C05458=1037.244,431.562,355.242,175.283,46.593,159.539
C05459=1037.232,431.317,355.292,175.268,46.586,159.535
C05460=1037.220,431.072,355.342,175.254,46.579,159.532
C05461=1037.208,430.829,355.393,175.240,46.572,159.528
C05462=1037.196,430.584,355.443,175.226,46.565,159.524
C05463=1037.184,430.339,355.494,175.213,46.558,159.521
C05464=1037.173,430.095,355.544,175.199,46.551,159.517
C05465=1037.161,429.850,355.594,175.184,46.544,159.513
C05466=1037.149,429.606,355.644,175.171,46.537,159.510
C05467=1037.138,429.360,355.694,175.157,46.530,159.506
C05468=1037.125,429.116,355.744,175.144,46.523,159.502
C05469=1037.114,428.871,355.793,175.130,46.516,159.499
C05470=1037.103,428.626,355.844,175.117,46.509,159.495
C05471=1037.091,428.382,355.894,175.103,46.503,159.492
C05472=1037.080,428.137,355.944,175.090,46.495,159.488
C05473=1037.068,427.892,355.994,175.076,46.489,159.485
C05474=1037.056,427.648,356.043,175.063,46.482,159.481
C05475=1037.044,427.402,356.093,175.049,46.475,159.478
C05476=1037.033,427.157,356.142,175.036,46.468,159.474
C05477=1037.022,426.913,356.192,175.023,46.462,159.471
C05478=1037.010,426.668,356.241,175.010,46.455,159.467
C05479=1036.998,426.423,356.290,174.997,46.448,159.464
C05480=1036.987,426.178,356.339,174.984,46.442,159.460
C05481=1036.975,425.933,356.389,174.970,46.435,159.457
C05482=1036.963,425.689,356.439,174.957,46.428,159.453
C05483=1036.952,425.444,356.488,174.944,46.422,159.450
C05484=1036.941,425.199,356.537,174.932,46.415,159.447
C05485=1036.930,424.953,356.585,174.919,46.409,159.443
C05486=1036.918,424.709,356.634,174.905,46.402,159.440
C05487=1036.907,424.464,356.684,174.892,46.395,159.436
C05488=1036.896,424.219,356.733,174.880,46.389,159.433
C05489=1036.884,423.974,356.782,174.867,46.383,159.430
C05490=1036.873,423.730,356.831,174.855,46.376,159.427
C05491=1036.861,423.484,356.879,174.842,46.370,159.423
C05492=1036.850,423.239,356.928,174.830,46.364,159.420
C05493=1036.839,423.000,356.976,174.817,46.357,159.417
C05494=1036.828,422.760,357.023,174.805,46.351,159.414
C05495=1036.817,422.521,357.070,174.793,46.345,159.411
C05496=1036.806,422.281,357.118,174.781,46.339,159.408
C05497=1036.795,422.041,357.165,174.769,46.333,159.404
C05498=1036.784,421.802,357.212,174.756,46.326,159.401
C05499=1036.774,421.562,357.259,174.745,46.320,159.398
C05500=1036.763,421.322,357.307,174.732,46.314,159.395
C05501=1036.752,421.077,357.355,174.720,46.308,159.392
C05502=1036.740,420.833,357.402,174.708,46.302,159.389
C05503=1036.729,420.588,357.451,174.696,46.296,159.386
C05504=1036.718,420.343,357.500,174.684,46.290,159.382
C05505=1036.708,420.097,357.547,174.672,46.283,159.379
C05506=1036.697,419.852,357.595,174.659,46.278,159.376
C05507=1036.685,419.607,357.644,174.648,46.271,159.373
C05508=1036.675,419.362,357.691,174.636,46.265,159.370
C05509=1036.664,419.117,357.740,174.623,46.259,159.367
C05510=1036.653,418.871,357.788,174.612,46.253,159.364
C05511=1036.642,418.626,357.835,174.600,46.247,159.361
C05512=1036.631,418.381,357.883,174.589,46.241,159.358
C05513=1036.620,418.136,357.931,174.576,46.235,159.355
C05514=1036.610,417.891,357.978,174.565,46.229,159.352
C05515=1036.599,417.646,358.026,174.553,46.223,159.349
C05516=1036.589,417.400,358.074,174.541,46.217,159.346
C05517=1036.577,417.155,358.121,174.530,46.211,159.343
C05518=1036.567,416.910,358.169,174.518,46.205,159.340
C05519=1036.556,416.664,358.216,174.507,46.200,159.337
C05520=1036.545,416.419,358.263,174.496,46.194,159.334
C05521=1036.535,416.174,358.311,174.484,46.188,159.331
C05522=1036.523,415.929,358.358,174.473,46.182,159.328
C05523=1036.513,415.683,358.405,174.461,46.177,159.325
C05524=1036.503,415.438,358.452,174.450,46.171,159.322
C05525=1036.491,415.192,358.499,174.439,46.165,159.320
C05526=1036.481,414.947,358.546,174.427,46.160,159.317
C05527=1036.470,414.702,358.593,174.416,46.154,159.314
C05528=1036.460,414.457,358.640,174.405,46.148,159.311
C05529=1036.450,414.212,358.687,174.393,46.142,159.308
C05530=1036.438,413.965,358.734,174.382,46.137,159.305
C05531=1036.428,413.720,358.781,174.371,46.131,159.303
C05532=1036.417,413.475,358.827,174.360,46.126,159.300
C05533=1036.407,413.230,358.875,174.349,46.120,159.297
C05534=1036.397,412.984,358.921,174.337,46.114,159.294
C05535=1036.386,412.739,358.968,174.327,46.109,159.291
C05536=1036.376,412.494,359.015,174.316,46.103,159.289
C05537=1036.365,412.248,359.061,174.305,46.098,159.286
C05538=1036.355,412.003,359.108,174.294,46.093,159.283
C05539=1036.345,411.757,359.155,174.284,46.087,159.281
C05540=1036.334,411.512,359.201,174.272,46.082,159.278
C05541=1036.325,411.266,359.248,174.261,46.076,159.275
C05542=1036.314,411.020,359.294,174.250,46.070,159.272
C05543=1036.303,410.775,359.340,174.240,46.065,159.270
C05544=1036.293,410.529,359.386,174.229,46.060,159.267
C05545=1036.283,410.285,359.432,174.218,46.055,159.264
C05546=1036.272,410.039,359.478,174.208,46.049,159.262
C05547=1036.262,409.793,359.524,174.197,46.044,159.259
C05548=1036.252,409.547,359.571,174.186,46.039,159.256
C05549=1036.241,409.302,359.617,174.176,46.034,159.254
C05550=1036.231,409.057,359.662,174.165,46.028,159.251
C05551=1036.221,408.811,359.707,174.155,46.023,159.249
C05552=1036.211,408.565,359.754,174.145,46.018,159.246
C05553=1036.201,408.330,359.798,174.135,46.013,159.244
C05554=1036.192,408.095,359.841,174.124,46.008,159.241
C05555=1036.181,407.860,359.886,174.115,46.003,159.239
C05556=1036.172,407.624,359.929,174.105,45.998,159.236
C05557=1036.162,407.390,359.972,174.095,45.993,159.234
C05558=1036.152,407.155,360.016,174.085,45.988,159.231
C05559=1036.144,406.919,360.060,174.076,45.983,159.229
C05560=1036.133,406.683,360.104,174.065,45.979,159.227
C05561=1036.123,406.439,360.150,174.056,45.973,159.224
C05562=1036.113,406.192,360.195,174.045,45.968,159.222
C05563=1036.103,405.947,360.240,174.035,45.963,159.219
C05564=1036.093,405.701,360.286,174.025,45.959,159.217
C05565=1036.084,405.455,360.331,174.015,45.953,159.214
C05566=1036.074,405.211,360.377,174.005,45.948,159.212
C05567=1036.063,404.964,360.422,173.995,45.944,159.209
C05568=1036.054,404.719,360.467,173.985,45.938,159.207
C05569=1036.044,404.474,360.513,173.975,45.933,159.204
C05570=1036.034,404.227,360.558,173.964,45.929,159.202
C05571=1036.024,403.982,360.603,173.955,45.923,159.199
C05572=1036.015,403.736,360.648,173.945,45.919,159.197
C05573=1036.005,403.490,360.693,173.936,45.914,159.195
C05574=1035.995,403.244,360.738,173.925,45.909,159.192
C05575=1035.986,402.999,360.783,173.916,45.904,159.190
C05576=1035.976,402.753,360.828,173.906,45.899,159.188
C05577=1035.966,402.508,360.873,173.896,45.894,159.185
C05578=1035.956,402.262,360.918,173.886,45.889,159.183
C05579=1035.946,402.016,360.963,173.877,45.885,159.181
C05580=1035.936,401.771,361.007,173.867,45.880,159.178
C05581=1035.927,401.525,361.052,173.858,45.875,159.176
C05582=1035.917,401.279,361.096,173.848,45.871,159.174
C05583=1035.908,401.033,361.141,173.838,45.866,159.171
C05584=1035.898,400.788,361.186,173.828,45.861,159.169
C05585=1035.889,400.542,361.230,173.819,45.856,159.167
C05586=1035.879,400.296,361.275,173.809,45.852,159.164
C05587=1035.869,400.050,361.319,173.800,45.848,159.162
C05588=1035.860,399.805,361.364,173.791,45.843,159.160
C05589=1035.850,399.558,361.408,173.781,45.838,159.158
C05590=1035.841,399.313,361.453,173.772,45.833,159.155
C05591=1035.830,399.067,361.496,173.763,45.829,159.153
C05592=1035.821,398.822,361.541,173.753,45.825,159.151
C05593=1035.811,398.575,361.585,173.743,45.820,159.149
C05594=1035.802,398.329,361.629,173.735,45.815,159.146
C05595=1035.792,398.083,361.673,173.724,45.811,159.144
C05596=1035.783,397.838,361.717,173.716,45.807,159.142
C05597=1035.773,397.593,361.761,173.707,45.802,159.140
C05598=1035.764,397.346,361.806,173.697,45.798,159.138
C05599=1035.754,397.100,361.850,173.688,45.793,159.135
C05600=1035.744,396.854,361.893,173.679,45.789,159.133
C05601=1035.735,396.609,361.937,173.670,45.784,159.131
C05602=1035.726,396.363,361.981,173.661,45.780,159.129
C05603=1035.717,396.117,362.025,173.651,45.776,159.127
C05604=1035.706,395.871,362.069,173.642,45.772,159.125
C05605=1035.698,395.626,362.112,173.633,45.767,159.122
C05606=1035.688,395.379,362.157,173.624,45.762,159.120
C05607=1035.679,395.133,362.200,173.615,45.758,159.118
C05608=1035.670,394.888,362.243,173.606,45.754,159.116
C05609=1035.660,394.641,362.287,173.597,45.750,159.114
C05610=1035.651,394.396,362.331,173.588,45.745,159.112
C05611=1035.642,394.150,362.374,173.579,45.741,159.110
C05612=1035.632,393.903,362.418,173.570,45.737,159.108
C05613=1035.623,393.678,362.457,173.563,45.733,159.106
C05614=1035.616,393.453,362.497,173.554,45.729,159.104
C05615=1035.607,393.228,362.536,173.545,45.725,159.102
C05616=1035.598,393.003,362.576,173.538,45.722,159.100
C05617=1035.590,392.778,362.616,173.530,45.718,159.098
C05618=1035.581,392.553,362.655,173.522,45.714,159.097
C05619=1035.573,392.328,362.695,173.514,45.710,159.095
C05620=1035.565,392.103,362.735,173.506,45.706,159.093
C05621=1035.555,391.857,362.777,173.497,45.702,159.091
C05622=1035.546,391.611,362.821,173.489,45.698,159.089
C05623=1035.537,391.366,362.864,173.480,45.694,159.087
C05624=1035.528,391.120,362.907,173.471,45.690,159.085
C05625=1035.519,390.873,362.950,173.462,45.686,159.083
C05626=1035.510,390.627,362.993,173.454,45.682,159.081
C05627=1035.501,390.380,363.036,173.445,45.678,159.079
C05628=1035.491,390.135,363.078,173.436,45.674,159.077
C05629=1035.482,389.889,363.121,173.428,45.670,159.075
C05630=1035.473,389.642,363.164,173.419,45.667,159.073
C05631=1035.464,389.396,363.207,173.412,45.662,159.071
C05632=1035.455,389.150,363.250,173.403,45.658,159.069
C05633=1035.446,388.905,363.292,173.394,45.654,159.067
C05634=1035.436,388.658,363.335,173.386,45.651,159.065
C05635=1035.428,388.412,363.378,173.377,45.647,159.063
C05636=1035.419,388.166,363.420,173.369,45.642,159.061
C05637=1035.410,387.920,363.463,173.361,45.638,159.060
C05638=1035.401,387.674,363.505,173.353,45.635,159.058
C05639=1035.391,387.427,363.548,173.344,45.631,159.056
C05640=1035.383,387.181,363.591,173.335,45.627,159.054
C05641=1035.374,386.935,363.633,173.327,45.623,159.052
C05642=1035.365,386.689,363.675,173.320,45.620,159.050
C05643=1035.356,386.443,363.717,173.311,45.616,159.048
C05644=1035.346,386.197,363.759,173.303,45.612,159.046
C05645=1035.337,385.950,363.801,173.294,45.608,159.045
C05646=1035.328,385.704,363.844,173.287,45.605,159.043
C05647=1035.319,385.458,363.886,173.278,45.601,159.041
C05648=1035.311,385.211,363.928,173.270,45.597,159.039
C05649=1035.301,384.966,363.970,173.261,45.594,159.037
C05650=1035.292,384.719,364.012,173.254,45.590,159.036
C05651=1035.283,384.473,364.054,173.245,45.586,159.034
C05652=1035.274,384.226,364.095,173.237,45.583,159.032
C05653=1035.265,383.981,364.138,173.230,45.579,159.030
C05654=1035.256,383.734,364.180,173.221,45.576,159.028
C05655=1035.248,383.488,364.222,173.213,45.572,159.027
C05656=1035.239,383.241,364.264,173.206,45.568,159.025
C05657=1035.230,382.995,364.305,173.197,45.565,159.023
C05658=1035.222,382.749,364.347,173.190,45.561,159.021
C05659=1035.213,382.503,364.388,173.181,45.557,159.019
C05660=1035.204,382.257,364.430,173.173,45.554,159.018
C05661=1035.195,382.010,364.472,173.166,45.551,159.016
C05662=1035.186,381.764,364.514,173.157,45.547,159.014
C05663=1035.177,381.517,364.555,173.150,45.543,159.012
C05664=1035.170,381.271,364.597,173.142,45.540,159.011
C05665=1035.161,381.025,364.639,173.135,45.537,159.009
C05666=1035.152,380.779,364.681,173.126,45.533,159.007
C05667=1035.143,380.532,364.722,173.119,45.529,159.006
C05668=1035.135,380.286,364.763,173.111,45.526,159.004
C05669=1035.126,380.040,364.805,173.104,45.523,159.002
C05670=1035.117,379.793,364.846,173.095,45.519,159.001
C05671=1035.108,379.547,364.888,173.088,45.516,158.999
C05672=1035.100,379.301,364.929,173.080,45.512,158.997
C05673=1035.085,378.885,364.999,173.067,45.506,158.994
C05674=1035.071,378.470,365.069,173.054,45.501,158.992
C05675=1035.057,378.055,365.138,173.042,45.495,158.989
C05676=1035.043,377.640,365.208,173.029,45.490,158.986
C05677=1035.033,377.393,365.248,173.021,45.487,158.984
C05678=1035.025,377.147,365.289,173.014,45.483,158.983
C05679=1035.017,376.900,365.330,173.005,45.480,158.981
C05680=1035.008,376.653,365.372,172.998,45.477,158.980
C05681=1035.000,376.407,365.412,172.991,45.473,158.978
C05682=1034.990,376.160,365.453,172.983,45.470,158.976
C05683=1034.982,375.914,365.493,172.976,45.467,158.975
C05684=1034.974,375.667,365.534,172.968,45.464,158.973
C05685=1034.965,375.421,365.576,172.961,45.461,158.972
C05686=1034.956,375.175,365.616,172.954,45.457,158.970
C05687=1034.948,374.929,365.657,172.946,45.455,158.968
C05688=1034.939,374.682,365.698,172.939,45.451,158.967
C05689=1034.931,374.435,365.738,172.932,45.448,158.965
C05690=1034.922,374.189,365.778,172.924,45.445,158.964
C05691=1034.914,373.942,365.819,172.916,45.442,158.962
C05692=1034.906,373.696,365.860,172.909,45.439,158.961
C05693=1034.897,373.449,365.901,172.902,45.436,158.959
C05694=1034.889,373.202,365.940,172.895,45.433,158.957
C05695=1034.881,372.956,365.981,172.887,45.430,158.956
C05696=1034.872,372.709,366.022,172.880,45.426,158.954
C05697=1034.863,372.463,366.062,172.873,45.423,158.953
C05698=1034.855,372.217,366.103,172.866,45.421,158.951
C05699=1034.847,371.969,366.143,172.858,45.418,158.950
C05700=1034.839,371.723,366.184,172.851,45.414,158.948
C05701=1034.830,371.477,366.224,172.844,45.411,158.947
C05702=1034.822,371.231,366.264,172.837,45.408,158.945
C05703=1034.814,370.983,366.304,172.830,45.405,158.944
C05704=1034.806,370.737,366.345,172.823,45.402,158.942
C05705=1034.797,370.490,366.384,172.815,45.400,158.941
C05706=1034.789,370.244,366.425,172.809,45.397,158.939
C05707=1034.781,369.998,366.466,172.802,45.394,158.938
C05708=1034.773,369.751,366.505,172.795,45.391,158.936
C05709=1034.764,369.503,366.545,172.788,45.388,158.935
C05710=1034.756,369.257,366.585,172.781,45.385,158.933
C05711=1034.748,369.011,366.625,172.774,45.382,158.932
C05712=1034.740,368.764,366.665,172.766,45.379,158.930
C05713=1034.731,368.518,366.705,172.759,45.377,158.929
C05714=1034.723,368.271,366.745,172.752,45.374,158.928
C05715=1034.714,368.024,366.784,172.745,45.371,158.926
C05716=1034.706,367.777,366.824,172.739,45.368,158.925
C05717=1034.698,367.531,366.864,172.732,45.366,158.924
C05718=1034.689,367.284,366.904,172.725,45.363,158.922
C05719=1034.681,367.037,366.943,172.718,45.360,158.921
C05720=1034.673,366.791,366.983,172.711,45.357,158.919
C05721=1034.665,366.544,367.023,172.704,45.354,158.918
C05722=1034.657,366.297,367.062,172.698,45.351,158.916
C05723=1034.648,366.051,367.101,172.691,45.349,158.915
C05724=1034.641,365.804,367.141,172.684,45.346,158.914
C05725=1034.632,365.557,367.181,172.677,45.343,158.912
C05726=1034.624,365.310,367.220,172.670,45.340,158.911
C05727=1034.616,365.064,367.260,172.664,45.338,158.910
C05728=1034.607,364.817,367.299,172.657,45.335,158.908
C05729=1034.595,364.422,367.362,172.646,45.331,158.906
C05730=1034.582,364.028,367.425,172.635,45.327,158.904
C05731=1034.569,363.633,367.488,172.624,45.322,158.902
C05732=1034.557,363.238,367.551,172.614,45.318,158.899
C05733=1034.548,362.991,367.591,172.607,45.316,158.898
C05734=1034.540,362.745,367.630,172.600,45.313,158.897
C05735=1034.533,362.498,367.669,172.593,45.310,158.895
C05736=1034.524,362.251,367.708,172.587,45.308,158.894
C05737=1034.516,362.005,367.747,172.580,45.306,158.893
C05738=1034.509,361.757,367.787,172.573,45.303,158.892
C05739=1034.501,361.511,367.826,172.567,45.300,158.890
C05740=1034.492,361.264,367.864,172.561,45.297,158.889
C05741=1034.484,361.017,367.903,172.554,45.295,158.888
C05742=1034.477,360.770,367.943,172.548,45.293,158.886
C05743=1034.468,360.523,367.982,172.541,45.290,158.885
C05744=1034.461,360.277,368.020,172.534,45.288,158.884
C05745=1034.452,360.030,368.059,172.528,45.285,158.882
C05746=1034.444,359.783,368.098,172.521,45.283,158.881
C05747=1034.436,359.536,368.136,172.515,45.280,158.880
C05748=1034.428,359.289,368.175,172.509,45.278,158.879
C05749=1034.420,359.042,368.214,172.502,45.276,158.877
C05750=1034.412,358.795,368.253,172.495,45.273,158.876
C05751=1034.404,358.549,368.291,172.489,45.271,158.875
C05752=1034.396,358.302,368.330,172.482,45.269,158.874
C05753=1034.388,358.055,368.368,172.477,45.266,158.873
C05754=1034.380,357.808,368.407,172.470,45.264,158.871
C05755=1034.372,357.561,368.445,172.463,45.261,158.870
C05756=1034.365,357.314,368.484,172.457,45.259,158.869
C05757=1034.357,357.067,368.523,172.451,45.257,158.868
C05758=1034.349,356.821,368.562,172.445,45.254,158.866
C05759=1034.341,356.574,368.600,172.438,45.252,158.865
C05760=1034.333,356.326,368.639,172.432,45.250,158.864
C05761=1034.325,356.080,368.677,172.426,45.248,158.863
C05762=1034.318,355.832,368.715,172.420,45.245,158.861
C05763=1034.310,355.586,368.753,172.413,45.243,158.860
C05764=1034.301,355.339,368.791,172.407,45.241,158.859
C05765=1034.294,355.092,368.830,172.401,45.238,158.858
C05766=1034.285,354.845,368.868,172.395,45.236,158.857
C05767=1034.278,354.598,368.906,172.388,45.234,158.855
C05768=1034.270,354.351,368.944,172.382,45.232,158.854
C05769=1034.263,354.104,368.983,172.376,45.229,158.853
C05770=1034.254,353.857,369.021,172.370,45.228,158.852
C05771=1034.246,353.610,369.058,172.363,45.225,158.851
C05772=1034.239,353.363,369.096,172.358,45.223,158.850
C05773=1034.231,353.116,369.135,172.351,45.221,158.848
C05774=1034.223,352.869,369.172,172.345,45.219,158.847
C05775=1034.215,352.622,369.211,172.339,45.217,158.846
C05776=1034.207,352.375,369.248,172.333,45.214,158.845
C05777=1034.200,352.129,369.286,172.326,45.212,158.844
C05778=1034.192,351.881,369.324,172.321,45.210,158.843
C05779=1034.184,351.634,369.362,172.314,45.208,158.842
C05780=1034.177,351.387,369.400,172.308,45.206,158.840
C05781=1034.169,351.140,369.438,172.303,45.204,158.839
C05782=1034.161,350.893,369.475,172.296,45.202,158.838
C05783=1034.153,350.647,369.514,172.291,45.199,158.837
C05784=1034.146,350.399,369.552,172.284,45.198,158.836
C05785=1034.134,350.011,369.611,172.275,45.194,158.834
C05786=1034.121,349.622,369.670,172.266,45.191,158.833
C05787=1034.110,349.233,369.729,172.256,45.188,158.831
C05788=1034.097,348.844,369.788,172.246,45.185,158.829
C05789=1034.090,348.597,369.826,172.241,45.183,158.828
C05790=1034.082,348.351,369.864,172.235,45.181,158.827
C05791=1034.075,348.104,369.901,172.229,45.179,158.826
C05792=1034.067,347.857,369.938,172.223,45.177,158.825
C05793=1034.059,347.609,369.976,172.217,45.175,158.824
C05794=1034.051,347.362,370.013,172.211,45.173,158.823
C05795=1034.044,347.115,370.050,172.205,45.171,158.822
C05796=1034.036,346.868,370.087,172.200,45.169,158.820
C05797=1034.028,346.621,370.125,172.193,45.167,158.819
C05798=1034.021,346.374,370.162,172.188,45.165,158.818
C05799=1034.013,346.127,370.199,172.182,45.163,158.817
C05800=1034.005,345.880,370.237,172.176,45.161,158.816
C05801=1033.997,345.633,370.274,172.170,45.160,158.815
C05802=1033.990,345.386,370.312,172.165,45.158,158.814
C05803=1033.982,345.138,370.348,172.158,45.156,158.813
C05804=1033.975,344.891,370.385,172.153,45.154,158.812
C05805=1033.967,344.644,370.422,172.147,45.152,158.811
C05806=1033.960,344.397,370.460,172.142,45.151,158.810
C05807=1033.952,344.150,370.497,172.136,45.149,158.809
C05808=1033.945,343.902,370.534,172.130,45.147,158.808
C05809=1033.936,343.603,370.578,172.124,45.145,158.807
C05810=1033.926,343.303,370.624,172.116,45.143,158.806
C05811=1033.917,343.003,370.669,172.109,45.140,158.804
C05812=1033.908,342.703,370.713,172.103,45.138,158.803
C05813=1033.901,342.456,370.750,172.097,45.136,158.802
C05814=1033.893,342.209,370.786,172.091,45.134,158.801
C05815=1033.886,341.962,370.824,172.085,45.133,158.800
C05816=1033.878,341.715,370.861,172.080,45.131,158.799
C05817=1033.871,341.467,370.897,172.075,45.129,158.798
C05818=1033.863,341.220,370.935,172.068,45.127,158.797
C05819=1033.856,340.973,370.971,172.063,45.126,158.796
C05820=1033.849,340.725,371.008,172.057,45.124,158.795
C05821=1033.841,340.478,371.045,172.052,45.123,158.794
C05822=1033.833,340.231,371.081,172.046,45.120,158.793
C05823=1033.825,339.984,371.118,172.040,45.119,158.792
C05824=1033.818,339.737,371.154,172.035,45.118,158.791
C05825=1033.811,339.490,371.190,172.029,45.116,158.790
C05826=1033.803,339.242,371.227,172.024,45.114,158.789
C05827=1033.795,338.995,371.264,172.019,45.113,158.789
C05828=1033.788,338.748,371.300,172.012,45.111,158.787
C05829=1033.780,338.500,371.336,172.007,45.109,158.787
C05830=1033.774,338.253,371.372,172.002,45.108,158.786
C05831=1033.766,338.007,371.409,171.996,45.107,158.785
C05832=1033.758,337.759,371.446,171.991,45.104,158.784
C05833=1033.750,337.512,371.482,171.986,45.103,158.783
C05834=1033.743,337.265,371.518,171.980,45.102,158.782
C05835=1033.736,337.017,371.554,171.975,45.100,158.781
C05836=1033.729,336.770,371.591,171.969,45.098,158.780
C05837=1033.721,336.522,371.627,171.964,45.096,158.779
C05838=1033.714,336.275,371.663,171.958,45.095,158.778
C05839=1033.706,336.028,371.699,171.953,45.094,158.777
C05840=1033.699,335.781,371.735,171.948,45.092,158.776
C05841=1033.689,335.442,371.785,171.940,45.090,158.775
C05842=1033.679,335.103,371.835,171.933,45.088,158.774
C05843=1033.669,334.764,371.884,171.925,45.086,158.773
C05844=1033.659,334.424,371.934,171.918,45.084,158.771
C05845=1033.651,334.177,371.970,171.913,45.082,158.770
C05846=1033.644,333.930,372.006,171.907,45.081,158.770
C05847=1033.636,333.682,372.042,171.902,45.079,158.769
C05848=1033.629,333.434,372.077,171.896,45.078,158.768
C05849=1033.622,333.188,372.113,171.892,45.077,158.767
C05850=1033.614,332.941,372.149,171.886,45.075,158.766
C05851=1033.606,332.694,372.185,171.881,45.074,158.765
C05852=1033.599,332.446,372.220,171.875,45.073,158.764
C05853=1033.592,332.199,372.256,171.870,45.071,158.764
C05854=1033.584,331.952,372.292,171.865,45.069,158.763
C05855=1033.577,331.703,372.328,171.860,45.068,158.762
C05856=1033.570,331.457,372.364,171.854,45.067,158.761
C05857=1033.563,331.209,372.399,171.849,45.066,158.760
C05858=1033.555,330.962,372.435,171.844,45.064,158.759
C05859=1033.548,330.714,372.470,171.839,45.063,158.758
C05860=1033.541,330.467,372.506,171.834,45.061,158.758
C05861=1033.533,330.220,372.543,171.829,45.060,158.757
C05862=1033.526,329.973,372.577,171.823,45.059,158.756
C05863=1033.518,329.725,372.613,171.818,45.057,158.755
C05864=1033.511,329.478,372.648,171.813,45.056,158.754
C05865=1033.505,329.230,372.684,171.808,45.055,158.754
C05866=1033.497,328.983,372.720,171.803,45.053,158.753
C05867=1033.490,328.736,372.755,171.798,45.052,158.752
C05868=1033.483,328.488,372.791,171.792,45.051,158.751
C05869=1033.476,328.241,372.826,171.787,45.050,158.750
C05870=1033.468,327.993,372.861,171.782,45.048,158.749
C05871=1033.461,327.746,372.896,171.777,45.047,158.749
C05872=1033.453,327.499,372.932,171.772,45.046,158.748
C05873=1033.446,327.251,372.967,171.767,45.045,158.747
C05874=1033.438,327.004,373.002,171.761,45.043,158.746
C05875=1033.431,326.756,373.037,171.756,45.043,158.745
C05876=1033.423,326.509,373.072,171.751,45.041,158.745
C05877=1033.416,326.261,373.107,171.746,45.040,158.744
C05878=1033.408,326.014,373.142,171.742,45.039,158.743
C05879=1033.402,325.767,373.177,171.737,45.038,158.742
C05880=1033.394,325.519,373.212,171.732,45.037,158.742
C05881=1033.387,325.271,373.247,171.727,45.035,158.741
C05882=1033.379,325.024,373.281,171.721,45.034,158.740
C05883=1033.372,324.776,373.317,171.716,45.034,158.739
C05884=1033.364,324.529,373.351,171.711,45.032,158.738
C05885=1033.358,324.282,373.387,171.706,45.031,158.738
C05886=1033.350,324.034,373.421,171.701,45.030,158.737
C05887=1033.343,323.787,373.457,171.696,45.029,158.736
C05888=1033.335,323.540,373.491,171.691,45.028,158.735
C05889=1033.328,323.293,373.526,171.687,45.027,158.735
C05890=1033.320,323.045,373.561,171.682,45.026,158.734
C05891=1033.313,322.798,373.596,171.677,45.024,158.733
C05892=1033.306,322.550,373.630,171.672,45.023,158.732
C05893=1033.299,322.303,373.665,171.666,45.023,158.732
C05894=1033.292,322.054,373.700,171.661,45.022,158.731
C05895=1033.284,321.807,373.735,171.656,45.020,158.730
C05896=1033.277,321.560,373.770,171.651,45.019,158.729
C05897=1033.266,321.164,373.824,171.644,45.017,158.728
C05898=1033.254,320.767,373.881,171.636,45.016,158.727
C05899=1033.243,320.371,373.936,171.628,45.014,158.726
C05900=1033.231,319.974,373.991,171.621,45.013,158.725
C05901=1033.224,319.726,374.026,171.616,45.012,158.724
C05902=1033.217,319.479,374.061,171.611,45.011,158.723
C05903=1033.210,319.231,374.095,171.607,45.010,158.723
C05904=1033.203,318.984,374.130,171.601,45.008,158.722
C05905=1033.196,318.736,374.164,171.597,45.007,158.721
C05906=1033.189,318.489,374.199,171.592,45.006,158.720
C05907=1033.181,318.242,374.233,171.587,45.005,158.720
C05908=1033.175,317.994,374.267,171.582,45.004,158.719
C05909=1033.167,317.747,374.302,171.577,45.004,158.718
C05910=1033.161,317.499,374.336,171.573,45.003,158.718
C05911=1033.153,317.252,374.371,171.568,45.002,158.717
C05912=1033.146,317.004,374.405,171.563,45.001,158.716
C05913=1033.139,316.756,374.439,171.558,45.000,158.716
C05914=1033.132,316.509,374.474,171.553,44.999,158.715
C05915=1033.125,316.261,374.508,171.549,44.998,158.714
C05916=1033.118,316.014,374.543,171.544,44.997,158.713
C05917=1033.112,315.766,374.577,171.539,44.996,158.713
C05918=1033.104,315.519,374.611,171.534,44.995,158.712
C05919=1033.097,315.272,374.645,171.529,44.994,158.711
C05920=1033.090,315.024,374.680,171.525,44.993,158.711
C05921=1033.083,314.776,374.714,171.521,44.992,158.710
C05922=1033.077,314.529,374.749,171.516,44.992,158.709
C05923=1033.070,314.282,374.782,171.511,44.991,158.709
C05924=1033.063,314.034,374.816,171.506,44.990,158.708
C05925=1033.056,313.787,374.851,171.502,44.989,158.707
C05926=1033.049,313.539,374.885,171.497,44.988,158.707
C05927=1033.041,313.291,374.919,171.492,44.987,158.706
C05928=1033.036,313.044,374.953,171.488,44.986,158.705
C05929=1033.028,312.796,374.987,171.484,44.985,158.705
C05930=1033.022,312.549,375.022,171.479,44.984,158.704
C05931=1033.014,312.301,375.056,171.474,44.984,158.703
C05932=1033.007,312.054,375.090,171.469,44.983,158.703
C05933=1033.001,311.806,375.124,171.464,44.982,158.702
C05934=1032.994,311.559,375.157,171.460,44.981,158.701
C05935=1032.987,311.311,375.191,171.456,44.980,158.701
C05936=1032.980,311.063,375.225,171.451,44.979,158.700
C05937=1032.973,310.816,375.259,171.447,44.979,158.700
C05938=1032.965,310.568,375.293,171.442,44.978,158.699
C05939=1032.958,310.321,375.326,171.437,44.978,158.698
C05940=1032.951,310.073,375.359,171.433,44.977,158.698
C05941=1032.944,309.825,375.393,171.428,44.976,158.697
C05942=1032.937,309.578,375.426,171.423,44.975,158.696
C05943=1032.929,309.330,375.460,171.419,44.975,158.696
C05944=1032.922,309.083,375.493,171.415,44.974,158.695
C05945=1032.915,308.835,375.526,171.410,44.973,158.695
C05946=1032.908,308.587,375.560,171.405,44.973,158.694
C05947=1032.901,308.340,375.594,171.401,44.972,158.693
C05948=1032.894,308.092,375.626,171.396,44.971,158.693
C05949=1032.887,307.845,375.660,171.392,44.971,158.692
C05950=1032.879,307.597,375.694,171.387,44.971,158.692
C05951=1032.873,307.349,375.727,171.383,44.969,158.691
C05952=1032.865,307.102,375.760,171.379,44.969,158.690
C05953=1032.854,306.710,375.812,171.372,44.968,158.690
C05954=1032.843,306.318,375.866,171.364,44.967,158.689
C05955=1032.832,305.927,375.918,171.358,44.966,158.688
C05956=1032.820,305.536,375.971,171.351,44.965,158.687
C05957=1032.814,305.287,376.004,171.346,44.964,158.686
C05958=1032.807,305.041,376.037,171.341,44.964,158.686
C05959=1032.799,304.793,376.070,171.337,44.964,158.685
C05960=1032.793,304.546,376.103,171.332,44.963,158.685
C05961=1032.786,304.297,376.136,171.328,44.962,158.684
C05962=1032.779,304.049,376.169,171.324,44.962,158.683
C05963=1032.772,303.802,376.202,171.319,44.961,158.683
C05964=1032.765,303.554,376.235,171.314,44.960,158.682
C05965=1032.758,303.307,376.269,171.311,44.960,158.682
C05966=1032.751,303.059,376.302,171.306,44.959,158.681
C05967=1032.744,302.811,376.334,171.302,44.959,158.681
C05968=1032.737,302.564,376.368,171.297,44.958,158.680
C05969=1032.731,302.316,376.401,171.293,44.958,158.679
C05970=1032.724,302.068,376.434,171.289,44.957,158.679
C05971=1032.716,301.821,376.467,171.284,44.957,158.678
C05972=1032.710,301.573,376.500,171.280,44.957,158.678
C05973=1032.703,301.325,376.533,171.276,44.955,158.677
C05974=1032.696,301.078,376.566,171.271,44.955,158.677
C05975=1032.689,300.830,376.599,171.267,44.955,158.676
C05976=1032.682,300.582,376.632,171.263,44.954,158.676
C05977=1032.676,300.335,376.664,171.259,44.954,158.675
C05978=1032.668,300.087,376.698,171.254,44.953,158.674
C05979=1032.662,299.840,376.730,171.249,44.952,158.674
C05980=1032.655,299.591,376.763,171.246,44.952,158.673
C05981=1032.648,299.344,376.796,171.241,44.952,158.673
C05982=1032.641,299.096,376.829,171.237,44.951,158.672
C05983=1032.634,298.848,376.861,171.233,44.951,158.672
C05984=1032.628,298.600,376.894,171.229,44.950,158.671
C05985=1032.621,298.353,376.928,171.224,44.950,158.671
C05986=1032.614,298.106,376.960,171.221,44.949,158.670
C05987=1032.607,297.857,376.993,171.216,44.948,158.670
C05988=1032.601,297.610,377.026,171.211,44.948,158.669
C05989=1032.594,297.362,377.058,171.208,44.947,158.669
C05990=1032.587,297.114,377.091,171.203,44.947,158.668
C05991=1032.581,296.866,377.124,171.199,44.947,158.667
C05992=1032.574,296.619,377.156,171.195,44.946,158.667
C05993=1032.567,296.371,377.189,171.190,44.946,158.666
C05994=1032.560,296.123,377.222,171.187,44.945,158.666
C05995=1032.554,295.876,377.255,171.182,44.945,158.665
C05996=1032.547,295.628,377.287,171.178,44.945,158.665
C05997=1032.540,295.380,377.320,171.174,44.944,158.664
C05998=1032.534,295.133,377.353,171.170,44.944,158.664
C05999=1032.527,294.885,377.385,171.165,44.943,158.663
C06000=1032.520,294.636,377.417,171.162,44.943,158.663
C06001=1032.513,294.389,377.449,171.157,44.942,158.662
C06002=1032.507,294.141,377.482,171.153,44.942,158.662
C06003=1032.499,293.893,377.515,171.149,44.942,158.661
C06004=1032.493,293.645,377.547,171.145,44.942,158.661
C06005=1032.486,293.398,377.579,171.141,44.941,158.660
C06006=1032.479,293.151,377.611,171.137,44.941,158.660
C06007=1032.473,292.902,377.643,171.132,44.940,158.659
C06008=1032.466,292.655,377.676,171.129,44.940,158.659
C06009=1032.455,292.280,377.725,171.122,44.940,158.658
C06010=1032.445,291.906,377.773,171.116,44.939,158.658
C06011=1032.434,291.531,377.821,171.110,44.939,158.657
C06012=1032.424,291.157,377.870,171.104,44.939,158.656
C06013=1032.417,290.908,377.902,171.099,44.938,158.656
C06014=1032.410,290.661,377.934,171.096,44.938,158.655
C06015=1032.404,290.413,377.966,171.091,44.938,158.655
C06016=1032.397,290.165,377.998,171.088,44.937,158.654
C06017=1032.390,289.917,378.030,171.083,44.938,158.654
C06018=1032.383,289.669,378.061,171.079,44.937,158.653
C06019=1032.377,289.421,378.094,171.075,44.937,158.653
C06020=1032.370,289.173,378.126,171.071,44.937,158.653
C06021=1032.363,288.926,378.158,171.068,44.936,158.652
C06022=1032.356,288.678,378.189,171.063,44.936,158.652
C06023=1032.349,288.430,378.221,171.060,44.936,158.651
C06024=1032.342,288.182,378.253,171.055,44.936,158.651
C06025=1032.336,287.934,378.285,171.051,44.936,158.650
C06026=1032.329,287.686,378.316,171.047,44.935,158.650
C06027=1032.322,287.439,378.349,171.043,44.936,158.649
C06028=1032.315,287.191,378.380,171.039,44.935,158.649
C06029=1032.309,286.943,378.412,171.035,44.935,158.648
C06030=1032.301,286.695,378.444,171.032,44.935,158.648
C06031=1032.295,286.447,378.476,171.027,44.934,158.648
C06032=1032.288,286.199,378.507,171.024,44.934,158.647
C06033=1032.281,285.951,378.539,171.019,44.934,158.647
C06034=1032.275,285.703,378.570,171.016,44.934,158.646
C06035=1032.268,285.456,378.602,171.012,44.934,158.646
C06036=1032.260,285.208,378.633,171.007,44.934,158.646
C06037=1032.254,284.960,378.665,171.004,44.934,158.645
C06038=1032.247,284.713,378.696,170.999,44.934,158.645
C06039=1032.240,284.465,378.728,170.996,44.934,158.644
C06040=1032.233,284.216,378.759,170.991,44.933,158.644
C06041=1032.226,283.968,378.791,170.988,44.933,158.644
C06042=1032.219,283.720,378.822,170.984,44.934,158.643
C06043=1032.213,283.472,378.854,170.980,44.933,158.643
C06044=1032.206,283.224,378.885,170.976,44.933,158.642
C06045=1032.199,282.977,378.917,170.973,44.933,158.642
C06046=1032.192,282.729,378.948,170.968,44.933,158.641
C06047=1032.186,282.481,378.979,170.965,44.933,158.641
C06048=1032.179,282.233,379.011,170.960,44.933,158.641
C06049=1032.172,281.985,379.042,170.957,44.933,158.640
C06050=1032.166,281.737,379.074,170.953,44.933,158.640
C06051=1032.158,281.489,379.105,170.949,44.932,158.639
C06052=1032.151,281.242,379.136,170.945,44.933,158.639
C06053=1032.145,280.994,379.167,170.942,44.933,158.639
C06054=1032.138,280.745,379.198,170.937,44.932,158.638
C06055=1032.131,280.497,379.230,170.934,44.932,158.638
C06056=1032.125,280.249,379.261,170.929,44.933,158.638
C06057=1032.118,280.001,379.292,170.926,44.933,158.637
C06058=1032.111,279.754,379.324,170.922,44.932,158.637
C06059=1032.105,279.506,379.355,170.918,44.932,158.636
C06060=1032.099,279.258,379.386,170.914,44.933,158.636
C06061=1032.092,279.010,379.417,170.911,44.932,158.636
C06062=1032.085,278.762,379.449,170.907,44.932,158.635
C06063=1032.078,278.514,379.479,170.903,44.932,158.635
C06064=1032.071,278.266,379.511,170.900,44.932,158.635
C06065=1032.062,277.903,379.557,170.894,44.932,158.634
C06066=1032.052,277.541,379.602,170.889,44.932,158.633
C06067=1032.042,277.178,379.647,170.883,44.933,158.633
C06068=1032.032,276.816,379.692,170.878,44.933,158.632
C06069=1032.025,276.568,379.722,170.873,44.933,158.632
C06070=1032.018,276.320,379.754,170.870,44.933,158.632
C06071=1032.012,276.072,379.785,170.866,44.933,158.631
C06072=1032.004,275.824,379.815,170.862,44.933,158.631
C06073=1031.999,275.576,379.846,170.858,44.933,158.630
C06074=1031.992,275.329,379.877,170.855,44.933,158.630
C06075=1031.985,275.080,379.907,170.851,44.933,158.630
C06076=1031.978,274.832,379.939,170.847,44.933,158.629
C06077=1031.971,274.584,379.970,170.844,44.933,158.629
C06078=1031.964,274.336,380.000,170.839,44.933,158.629
C06079=1031.958,274.088,380.031,170.836,44.933,158.628
C06080=1031.951,273.841,380.062,170.832,44.934,158.628
C06081=1031.944,273.592,380.092,170.829,44.934,158.628
C06082=1031.938,273.344,380.123,170.825,44.934,158.627
C06083=1031.930,273.096,380.154,170.821,44.934,158.627
C06084=1031.925,272.848,380.184,170.818,44.934,158.627
C06085=1031.918,272.600,380.215,170.813,44.934,158.626
C06086=1031.911,272.352,380.246,170.810,44.934,158.626
C06087=1031.904,272.104,380.276,170.807,44.934,158.626
C06088=1031.897,271.856,380.307,170.803,44.935,158.625
C06089=1031.891,271.608,380.338,170.799,44.935,158.625
C06090=1031.884,271.360,380.368,170.796,44.935,158.625
C06091=1031.877,271.112,380.398,170.792,44.935,158.624
C06092=1031.871,270.864,380.430,170.788,44.935,158.624
C06093=1031.864,270.616,380.460,170.784,44.935,158.624
C06094=1031.858,270.368,380.490,170.781,44.935,158.623
C06095=1031.851,270.119,380.521,170.778,44.935,158.623
C06096=1031.844,269.872,380.550,170.773,44.936,158.623
C06097=1031.837,269.624,380.582,170.770,44.936,158.623
C06098=1031.830,269.376,380.612,170.767,44.936,158.622
C06099=1031.824,269.127,380.643,170.763,44.937,158.622
C06100=1031.817,268.880,380.672,170.759,44.937,158.621
C06101=1031.810,268.632,380.702,170.756,44.937,158.621
C06102=1031.804,268.383,380.733,170.752,44.937,158.621
C06103=1031.797,268.136,380.763,170.748,44.937,158.620
C06104=1031.791,267.887,380.794,170.744,44.938,158.620
C06105=1031.784,267.639,380.824,170.741,44.938,158.620
C06106=1031.777,267.391,380.853,170.738,44.938,158.620
C06107=1031.771,267.143,380.884,170.734,44.938,158.619
C06108=1031.763,266.895,380.914,170.730,44.938,158.619
C06109=1031.758,266.647,380.945,170.727,44.939,158.619
C06110=1031.750,266.399,380.975,170.723,44.939,158.618
C06111=1031.743,266.150,381.005,170.720,44.939,158.618
C06112=1031.737,265.903,381.035,170.716,44.939,158.618
C06113=1031.730,265.654,381.065,170.712,44.940,158.618
C06114=1031.723,265.406,381.096,170.709,44.940,158.617
C06115=1031.717,265.159,381.125,170.706,44.940,158.617
C06116=1031.709,264.910,381.155,170.701,44.940,158.617
C06117=1031.704,264.663,381.186,170.698,44.941,158.616
C06118=1031.696,264.414,381.216,170.695,44.941,158.616
C06119=1031.690,264.165,381.245,170.691,44.941,158.616
C06120=1031.683,263.918,381.275,170.688,44.942,158.616
C06121=1031.673,263.560,381.319,170.682,44.943,158.615
C06122=1031.664,263.202,381.362,170.678,44.943,158.615
C06123=1031.654,262.844,381.405,170.673,44.943,158.614
C06124=1031.645,262.487,381.449,170.668,44.944,158.614
C06125=1031.638,262.238,381.478,170.664,44.944,158.614
C06126=1031.631,261.990,381.508,170.661,44.944,158.613
C06127=1031.624,261.742,381.538,170.657,44.945,158.613
C06128=1031.618,261.494,381.569,170.654,44.945,158.613
C06129=1031.612,261.246,381.598,170.650,44.945,158.612
C06130=1031.605,260.998,381.628,170.646,44.946,158.612
C06131=1031.598,260.749,381.657,170.643,44.946,158.612
C06132=1031.590,260.501,381.686,170.640,44.946,158.612
C06133=1031.584,260.253,381.715,170.636,44.947,158.611
C06134=1031.577,260.005,381.746,170.633,44.947,158.611
C06135=1031.570,259.756,381.775,170.630,44.948,158.611
C06136=1031.564,259.509,381.805,170.625,44.948,158.611
C06137=1031.557,259.260,381.834,170.622,44.949,158.611
C06138=1031.549,259.013,381.863,170.619,44.949,158.610
C06139=1031.543,258.764,381.893,170.616,44.950,158.610
C06140=1031.536,258.516,381.922,170.612,44.950,158.610
C06141=1031.529,258.268,381.952,170.609,44.951,158.610
C06142=1031.523,258.020,381.982,170.606,44.951,158.609
C06143=1031.516,257.771,382.011,170.601,44.951,158.609
C06144=1031.509,257.524,382.040,170.598,44.952,158.609
C06145=1031.502,257.275,382.070,170.595,44.952,158.609
C06146=1031.495,257.027,382.099,170.592,44.953,158.608
C06147=1031.488,256.779,382.129,170.588,44.953,158.608
C06148=1031.482,256.531,382.158,170.585,44.954,158.608
C06149=1031.475,256.282,382.187,170.582,44.954,158.608
C06150=1031.468,256.035,382.216,170.577,44.955,158.607
C06151=1031.461,255.786,382.246,170.574,44.955,158.607
C06152=1031.455,255.538,382.275,170.571,44.956,158.607
C06153=1031.448,255.290,382.305,170.568,44.956,158.607
C06154=1031.441,255.041,382.334,170.564,44.957,158.606
C06155=1031.435,254.793,382.363,170.561,44.957,158.606
C06156=1031.428,254.545,382.392,170.558,44.958,158.606
C06157=1031.421,254.297,382.422,170.554,44.958,158.606
C06158=1031.414,254.048,382.451,170.551,44.958,158.606
C06159=1031.408,253.800,382.480,170.547,44.959,158.605
C06160=1031.402,253.552,382.509,170.544,44.960,158.605
C06161=1031.394,253.304,382.539,170.541,44.960,158.605
C06162=1031.387,253.056,382.568,170.538,44.961,158.605
C06163=1031.381,252.808,382.597,170.534,44.961,158.604
C06164=1031.374,252.559,382.626,170.530,44.961,158.604
C06165=1031.368,252.311,382.655,170.527,44.962,158.604
C06166=1031.361,252.063,382.685,170.524,44.963,158.604
C06167=1031.354,251.815,382.714,170.521,44.963,158.604
C06168=1031.348,251.567,382.743,170.517,44.964,158.603
C06169=1031.341,251.318,382.772,170.514,44.964,158.603
C06170=1031.335,251.070,382.801,170.511,44.964,158.603
C06171=1031.328,250.822,382.830,170.508,44.965,158.603
C06172=1031.321,250.574,382.859,170.505,44.966,158.603
C06173=1031.315,250.325,382.888,170.500,44.966,158.602
C06174=1031.308,250.078,382.918,170.497,44.967,158.602
C06175=1031.302,249.829,382.947,170.494,44.967,158.602
C06176=1031.295,249.581,382.976,170.491,44.968,158.602
C06177=1031.286,249.222,383.017,170.486,44.968,158.601
C06178=1031.276,248.863,383.060,170.482,44.969,158.601
C06179=1031.267,248.503,383.102,170.477,44.970,158.601
C06180=1031.257,248.144,383.144,170.473,44.971,158.600
C06181=1031.250,247.896,383.173,170.468,44.972,158.600
C06182=1031.244,247.648,383.202,170.465,44.972,158.600
C06183=1031.237,247.399,383.231,170.462,44.972,158.600
C06184=1031.230,247.151,383.260,170.459,44.973,158.600
C06185=1031.224,246.903,383.289,170.456,44.974,158.599
C06186=1031.218,246.655,383.318,170.453,44.974,158.599
C06187=1031.212,246.406,383.346,170.450,44.974,158.599
C06188=1031.204,246.157,383.375,170.447,44.975,158.599
C06189=1031.198,245.909,383.404,170.443,44.976,158.599
C06190=1031.192,245.661,383.433,170.439,44.976,158.598
C06191=1031.186,245.413,383.462,170.436,44.977,158.598
C06192=1031.179,245.165,383.491,170.433,44.977,158.598
C06193=1031.172,244.917,383.520,170.430,44.978,158.598
C06194=1031.165,244.668,383.549,170.427,44.979,158.598
C06195=1031.159,244.419,383.577,170.424,44.979,158.597
C06196=1031.152,244.172,383.606,170.421,44.979,158.597
C06197=1031.146,243.923,383.635,170.418,44.980,158.597
C06198=1031.139,243.676,383.663,170.414,44.981,158.597
C06199=1031.133,243.427,383.692,170.411,44.982,158.597
C06200=1031.126,243.178,383.720,170.408,44.982,158.596
C06201=1031.119,242.930,383.749,170.405,44.983,158.596
C06202=1031.113,242.682,383.777,170.402,44.984,158.596
C06203=1031.107,242.434,383.806,170.399,44.984,158.596
C06204=1031.100,242.186,383.835,170.396,44.985,158.596
C06205=1031.094,241.937,383.863,170.393,44.986,158.596
C06206=1031.086,241.689,383.892,170.388,44.986,158.595
C06207=1031.080,241.440,383.921,170.385,44.986,158.595
C06208=1031.073,241.192,383.948,170.382,44.987,158.595
C06209=1031.067,240.944,383.978,170.379,44.988,158.595
C06210=1031.060,240.695,384.005,170.376,44.988,158.595
C06211=1031.054,240.447,384.034,170.373,44.989,158.594
C06212=1031.047,240.199,384.063,170.370,44.990,158.594
C06213=1031.041,239.951,384.091,170.367,44.990,158.594
C06214=1031.034,239.703,384.120,170.364,44.991,158.594
C06215=1031.027,239.454,384.148,170.360,44.992,158.594
C06216=1031.020,239.205,384.175,170.357,44.993,158.594
C06217=1031.014,238.957,384.204,170.354,44.994,158.594
C06218=1031.007,238.709,384.232,170.351,44.995,158.593
C06219=1031.000,238.461,384.261,170.348,44.995,158.593
C06220=1030.993,238.212,384.288,170.345,44.996,158.593
C06221=1030.987,237.964,384.317,170.342,44.997,158.593
C06222=1030.981,237.716,384.345,170.339,44.997,158.593
C06223=1030.974,237.467,384.373,170.336,44.998,158.593
C06224=1030.967,237.220,384.401,170.333,44.999,158.592
C06225=1030.960,236.970,384.430,170.329,45.000,158.592
C06226=1030.954,236.722,384.458,170.326,45.000,158.592
C06227=1030.947,236.474,384.486,170.323,45.001,158.592
C06228=1030.940,236.225,384.514,170.320,45.002,158.592
C06229=1030.933,235.977,384.542,170.317,45.003,158.592
C06230=1030.927,235.729,384.571,170.314,45.003,158.592
C06231=1030.920,235.480,384.598,170.311,45.004,158.591
C06232=1030.914,235.232,384.626,170.308,45.005,158.591
C06233=1030.904,234.866,384.667,170.303,45.006,158.591
C06234=1030.894,234.502,384.709,170.299,45.007,158.591
C06235=1030.884,234.136,384.750,170.294,45.009,158.591
C06236=1030.874,233.771,384.791,170.290,45.009,158.590
C06237=1030.869,233.523,384.819,170.287,45.010,158.590
C06238=1030.862,233.275,384.847,170.284,45.011,158.590
C06239=1030.855,233.027,384.875,170.281,45.012,158.590
C06240=1030.848,232.778,384.902,170.278,45.013,158.590
C06241=1030.842,232.530,384.930,170.275,45.013,158.590
C06242=1030.835,232.281,384.958,170.272,45.014,158.590
C06243=1030.829,232.033,384.987,170.268,45.015,158.589
C06244=1030.822,231.785,385.015,170.265,45.016,158.589
C06245=1030.815,231.536,385.042,170.262,45.017,158.589
C06246=1030.809,231.288,385.070,170.259,45.018,158.589
C06247=1030.802,231.039,385.098,170.256,45.018,158.589
C06248=1030.795,230.791,385.126,170.253,45.019,158.589
C06249=1030.789,230.542,385.153,170.250,45.020,158.589
C06250=1030.782,230.294,385.181,170.247,45.021,158.589
C06251=1030.775,230.046,385.209,170.244,45.022,158.589
C06252=1030.769,229.797,385.237,170.241,45.023,158.589
C06253=1030.762,229.549,385.264,170.238,45.024,158.588
C06254=1030.755,229.300,385.292,170.235,45.024,158.588
C06255=1030.749,229.052,385.320,170.232,45.025,158.588
C06256=1030.743,228.804,385.347,170.229,45.026,158.588
C06257=1030.736,228.556,385.375,170.226,45.027,158.588
C06258=1030.729,228.307,385.403,170.223,45.028,158.588
C06259=1030.723,228.059,385.430,170.221,45.029,158.588
C06260=1030.716,227.810,385.458,170.218,45.029,158.588
C06261=1030.709,227.562,385.486,170.214,45.030,158.587
C06262=1030.702,227.313,385.513,170.212,45.031,158.587
C06263=1030.696,227.064,385.540,170.209,45.032,158.587
C06264=1030.689,226.816,385.568,170.206,45.033,158.587
C06265=1030.683,226.568,385.595,170.203,45.034,158.587
C06266=1030.676,226.320,385.623,170.200,45.035,158.587
C06267=1030.669,226.072,385.650,170.197,45.036,158.587
C06268=1030.663,225.823,385.678,170.194,45.037,158.587
C06269=1030.655,225.574,385.705,170.191,45.037,158.587
C06270=1030.649,225.326,385.732,170.188,45.039,158.587
C06271=1030.642,225.078,385.760,170.185,45.039,158.586
C06272=1030.635,224.829,385.788,170.182,45.041,158.586
C06273=1030.629,224.581,385.814,170.179,45.041,158.586
C06274=1030.622,224.333,385.842,170.177,45.043,158.586
C06275=1030.616,224.084,385.869,170.173,45.043,158.586
C06276=1030.609,223.835,385.896,170.170,45.044,158.586
C06277=1030.602,223.587,385.924,170.168,45.045,158.586
C06278=1030.595,223.339,385.951,170.165,45.046,158.586
C06279=1030.589,223.091,385.979,170.162,45.047,158.586
C06280=1030.583,222.842,386.006,170.159,45.048,158.586
C06281=1030.576,222.593,386.033,170.156,45.049,158.586
C06282=1030.568,222.345,386.060,170.153,45.050,158.585
C06283=1030.562,222.096,386.087,170.150,45.051,158.585
C06284=1030.556,221.848,386.115,170.147,45.052,158.585
C06285=1030.550,221.599,386.142,170.144,45.053,158.585
C06286=1030.542,221.351,386.169,170.141,45.054,158.585
C06287=1030.536,221.103,386.197,170.138,45.055,158.585
C06288=1030.529,220.854,386.224,170.136,45.056,158.585
C06289=1030.519,220.481,386.265,170.131,45.058,158.585
C06290=1030.509,220.109,386.305,170.127,45.059,158.585
C06291=1030.500,219.736,386.346,170.123,45.060,158.585
C06292=1030.490,219.362,386.387,170.118,45.062,158.584
C06293=1030.483,219.115,386.414,170.115,45.062,158.584
C06294=1030.477,218.866,386.441,170.112,45.064,158.584
C06295=1030.469,218.618,386.468,170.109,45.064,158.584
C06296=1030.463,218.368,386.495,170.106,45.066,158.584
C06297=1030.456,218.121,386.522,170.104,45.067,158.584
C06298=1030.450,217.872,386.549,170.101,45.068,158.584
C06299=1030.443,217.623,386.575,170.098,45.069,158.584
C06300=1030.436,217.375,386.603,170.095,45.070,158.584
C06301=1030.429,217.127,386.629,170.092,45.071,158.584
C06302=1030.423,216.878,386.657,170.089,45.072,158.584
C06303=1030.416,216.630,386.683,170.086,45.073,158.584
C06304=1030.410,216.381,386.710,170.084,45.074,158.584
C06305=1030.402,216.133,386.737,170.082,45.075,158.584
C06306=1030.395,215.884,386.763,170.079,45.076,158.583
C06307=1030.389,215.635,386.790,170.076,45.077,158.583
C06308=1030.382,215.388,386.817,170.073,45.078,158.583
C06309=1030.376,215.139,386.844,170.070,45.079,158.583
C06310=1030.369,214.890,386.870,170.067,45.081,158.583
C06311=1030.363,214.642,386.897,170.064,45.081,158.583
C06312=1030.355,214.393,386.924,170.061,45.083,158.583
C06313=1030.349,214.144,386.951,170.059,45.084,158.583
C06314=1030.343,213.896,386.977,170.056,45.085,158.583
C06315=1030.336,213.648,387.005,170.053,45.086,158.583
C06316=1030.329,213.399,387.031,170.050,45.087,158.583
C06317=1030.323,213.151,387.058,170.047,45.088,158.583
C06318=1030.316,212.902,387.085,170.044,45.089,158.583
C06319=1030.310,212.654,387.112,170.042,45.090,158.583
C06320=1030.303,212.406,387.138,170.039,45.091,158.583
C06321=1030.296,212.157,387.165,170.037,45.092,158.583
C06322=1030.290,211.908,387.191,170.034,45.094,158.583
C06323=1030.283,211.660,387.218,170.031,45.094,158.583
C06324=1030.277,211.412,387.245,170.028,45.096,158.582
C06325=1030.269,211.163,387.272,170.025,45.096,158.582
C06326=1030.263,210.914,387.299,170.022,45.098,158.582
C06327=1030.257,210.666,387.325,170.019,45.099,158.582
C06328=1030.249,210.417,387.351,170.017,45.100,158.582
C06329=1030.244,210.169,387.378,170.014,45.101,158.582
C06330=1030.237,209.920,387.404,170.012,45.102,158.582
C06331=1030.229,209.672,387.431,170.009,45.103,158.582
C06332=1030.223,209.423,387.457,170.006,45.105,158.582
C06333=1030.217,209.174,387.484,170.003,45.105,158.582
C06334=1030.210,208.926,387.510,170.000,45.107,158.582
C06335=1030.203,208.678,387.536,169.998,45.108,158.582
C06336=1030.196,208.429,387.563,169.995,45.109,158.582
C06337=1030.190,208.180,387.589,169.992,45.110,158.582
C06338=1030.183,207.932,387.616,169.989,45.111,158.582
C06339=1030.176,207.684,387.642,169.986,45.112,158.582
C06340=1030.169,207.435,387.668,169.984,45.114,158.582
C06341=1030.163,207.187,387.694,169.982,45.115,158.582
C06342=1030.156,206.938,387.721,169.979,45.116,158.582
C06343=1030.150,206.690,387.747,169.976,45.117,158.582
C06344=1030.143,206.441,387.774,169.973,45.118,158.582
C06345=1030.133,206.074,387.813,169.969,45.120,158.582
C06346=1030.123,205.707,387.851,169.965,45.122,158.582
C06347=1030.113,205.340,387.890,169.961,45.124,158.582
C06348=1030.102,204.973,387.929,169.957,45.125,158.582
C06349=1030.073,203.714,388.054,169.595,45.023,158.524
C06350=1030.062,203.294,388.096,169.589,45.027,158.524
C06351=1030.056,203.046,388.121,169.585,45.028,158.524
C06352=1030.050,202.797,388.145,169.582,45.031,158.524
C06353=1030.044,202.549,388.170,169.578,45.033,158.524
C06354=1030.038,202.300,388.195,169.574,45.034,158.524
C06355=1030.033,202.052,388.220,169.571,45.037,158.524
C06356=1030.027,201.802,388.245,169.567,45.039,158.524
C06357=1030.020,201.554,388.270,169.563,45.040,158.524
C06358=1030.014,201.305,388.294,169.559,45.043,158.524
C06359=1030.008,201.057,388.319,169.555,45.045,158.524
C06360=1030.002,200.807,388.344,169.551,45.046,158.524
C06361=1029.997,200.559,388.368,169.548,45.048,158.524
C06362=1029.991,200.310,388.393,169.544,45.051,158.524
C06363=1029.984,200.061,388.417,169.541,45.053,158.524
C06364=1029.979,199.813,388.442,169.537,45.055,158.525
C06365=1029.972,199.564,388.466,169.533,45.057,158.524
C06366=1029.966,199.315,388.491,169.530,45.059,158.525
C06367=1029.960,199.067,388.515,169.526,45.061,158.525
C06368=1029.954,198.817,388.539,169.523,45.063,158.525
C06369=1029.947,198.569,388.564,169.519,45.065,158.525
C06370=1029.942,198.320,388.588,169.516,45.067,158.525
C06371=1029.935,198.071,388.612,169.512,45.070,158.525
C06372=1029.929,197.822,388.637,169.508,45.072,158.525
C06373=1029.923,197.574,388.660,169.505,45.074,158.525
C06374=1029.917,197.325,388.686,169.501,45.076,158.525
C06375=1029.911,197.077,388.709,169.498,45.078,158.525
C06376=1029.905,196.828,388.734,169.494,45.080,158.525
C06377=1029.898,196.579,388.758,169.490,45.082,158.525
C06378=1029.893,196.330,388.782,169.487,45.084,158.525
C06379=1029.887,196.081,388.806,169.483,45.086,158.526
C06380=1029.880,195.833,388.830,169.480,45.089,158.526
C06381=1029.874,195.584,388.855,169.476,45.091,158.526
C06382=1029.868,195.336,388.879,169.473,45.093,158.526
C06383=1029.862,195.087,388.904,169.469,45.095,158.526
C06384=1029.856,194.838,388.927,169.466,45.097,158.526
C06385=1029.850,194.589,388.952,169.462,45.100,158.526
C06386=1029.844,194.340,388.976,169.459,45.102,158.526
C06387=1029.838,194.091,389.000,169.455,45.104,158.526
C06388=1029.832,193.842,389.024,169.451,45.106,158.526
C06389=1029.827,193.594,389.049,169.448,45.108,158.526
C06390=1029.820,193.345,389.073,169.444,45.110,158.526
C06391=1029.815,193.096,389.097,169.441,45.112,158.526
C06392=1029.809,192.848,389.120,169.437,45.114,158.527
C06393=1029.802,192.599,389.145,169.433,45.116,158.527
C06394=1029.797,192.350,389.169,169.430,45.119,158.527
C06395=1029.790,192.101,389.193,169.426,45.121,158.527
C06396=1029.785,191.853,389.217,169.423,45.123,158.527
C06397=1029.778,191.604,389.241,169.419,45.125,158.527
C06398=1029.773,191.355,389.265,169.416,45.127,158.527
C06399=1029.765,191.015,389.298,169.411,45.130,158.527
C06400=1029.756,190.675,389.330,169.406,45.134,158.527
C06401=1029.748,190.335,389.363,169.401,45.136,158.527
C06402=1029.740,189.995,389.396,169.397,45.139,158.528
C06403=1029.735,189.746,389.420,169.394,45.141,158.528
C06404=1029.728,189.498,389.444,169.390,45.144,158.528
C06405=1029.722,189.249,389.468,169.386,45.146,158.528
C06406=1029.717,189.000,389.492,169.383,45.148,158.528
C06407=1029.710,188.716,389.519,169.379,45.150,158.528
C06408=1029.703,188.433,389.546,169.375,45.153,158.528
C06409=1029.696,188.150,389.574,169.371,45.155,158.528
C06410=1029.690,187.866,389.601,169.367,45.158,158.528
C06411=1029.684,187.618,389.624,169.364,45.160,158.528
C06412=1029.678,187.369,389.649,169.361,45.162,158.529
C06413=1029.672,187.120,389.673,169.357,45.164,158.529
C06414=1029.666,186.871,389.696,169.354,45.166,158.529
C06415=1029.660,186.622,389.720,169.350,45.169,158.529
C06416=1029.654,186.374,389.744,169.347,45.171,158.529
C06417=1029.649,186.125,389.767,169.343,45.174,158.529
C06418=1029.643,185.876,389.791,169.341,45.176,158.529
C06419=1029.637,185.627,389.816,169.337,45.178,158.529
C06420=1029.632,185.378,389.839,169.334,45.180,158.529
C06421=1029.626,185.130,389.862,169.330,45.182,158.530
C06422=1029.620,184.881,389.887,169.327,45.184,158.530
C06423=1029.614,184.632,389.910,169.323,45.187,158.530
C06424=1029.609,184.383,389.934,169.321,45.188,158.530
C06425=1029.603,184.135,389.958,169.317,45.191,158.530
C06426=1029.596,183.885,389.981,169.313,45.193,158.530
C06427=1029.591,183.637,390.005,169.310,45.195,158.530
C06428=1029.585,183.388,390.029,169.306,45.197,158.530
C06429=1029.580,183.139,390.053,169.304,45.199,158.530
C06430=1029.573,182.890,390.077,169.300,45.201,158.530
C06431=1029.568,182.641,390.100,169.297,45.204,158.530
C06432=1029.562,182.392,390.123,169.293,45.207,158.531
C06433=1029.555,182.143,390.147,169.290,45.209,158.531
C06434=1029.549,181.895,390.169,169.287,45.212,158.531
C06435=1029.543,181.647,390.193,169.283,45.214,158.531
C06436=1029.537,181.398,390.215,169.279,45.216,158.531
C06437=1029.531,181.148,390.239,169.277,45.219,158.532
C06438=1029.525,180.899,390.262,169.274,45.221,158.532
C06439=1029.518,180.651,390.285,169.270,45.223,158.532
C06440=1029.512,180.402,390.308,169.267,45.226,158.532
C06441=1029.506,180.153,390.331,169.263,45.228,158.532
C06442=1029.500,179.904,390.355,169.260,45.231,158.532
C06443=1029.494,179.656,390.378,169.256,45.233,158.532
C06444=1029.487,179.406,390.400,169.253,45.235,158.532
C06445=1029.482,179.157,390.423,169.251,45.238,158.533
C06446=1029.476,178.908,390.446,169.247,45.240,158.533
C06447=1029.470,178.660,390.470,169.244,45.243,158.533
C06448=1029.464,178.411,390.493,169.240,45.245,158.533
C06449=1029.457,178.162,390.516,169.237,45.247,158.533
C06450=1029.451,177.913,390.539,169.233,45.250,158.533
C06451=1029.446,177.664,390.562,169.230,45.252,158.534
C06452=1029.439,177.416,390.585,169.227,45.254,158.534
C06453=1029.434,177.167,390.608,169.224,45.257,158.534
C06454=1029.427,176.918,390.631,169.220,45.260,158.534
C06455=1029.421,176.669,390.654,169.217,45.262,158.534
C06456=1029.415,176.420,390.677,169.214,45.265,158.534
C06457=1029.409,176.171,390.700,169.211,45.267,158.535
C06458=1029.404,175.922,390.723,169.208,45.269,158.535
C06459=1029.397,175.674,390.746,169.204,45.272,158.535
C06460=1029.391,175.425,390.769,169.201,45.274,158.535
C06461=1029.385,175.176,390.792,169.197,45.277,158.535
C06462=1029.379,174.927,390.815,169.195,45.279,158.535
C06463=1029.373,174.678,390.837,169.191,45.282,158.535
C06464=1029.367,174.429,390.860,169.188,45.284,158.536
C06465=1029.361,174.180,390.883,169.185,45.287,158.536
C06466=1029.356,173.932,390.906,169.181,45.289,158.536
C06467=1029.350,173.683,390.929,169.179,45.291,158.536
C06468=1029.343,173.433,390.952,169.175,45.294,158.536
C06469=1029.337,173.184,390.975,169.172,45.296,158.536
C06470=1029.331,172.936,390.998,169.168,45.299,158.537
C06471=1029.325,172.652,391.024,169.165,45.302,158.537
C06472=1029.318,172.368,391.049,169.162,45.304,158.537
C06473=1029.311,172.085,391.075,169.157,45.307,158.537
C06474=1029.304,171.801,391.102,169.154,45.310,158.537
C06475=1029.298,171.552,391.125,169.150,45.312,158.537
C06476=1029.293,171.303,391.147,169.148,45.315,158.538
C06477=1029.286,171.054,391.169,169.145,45.317,158.538
C06478=1029.281,170.805,391.192,169.141,45.320,158.538
C06479=1029.275,170.556,391.215,169.139,45.322,158.538
C06480=1029.269,170.307,391.238,169.136,45.325,158.538
C06481=1029.263,170.059,391.260,169.132,45.327,158.538
C06482=1029.257,169.810,391.283,169.128,45.329,158.538
C06483=1029.251,169.561,391.306,169.126,45.332,158.539
C06484=1029.246,169.312,391.329,169.123,45.334,158.539
C06485=1029.239,169.063,391.352,169.119,45.337,158.539
C06486=1029.234,168.814,391.374,169.117,45.339,158.539
C06487=1029.228,168.565,391.397,169.113,45.342,158.539
C06488=1029.222,168.316,391.420,169.110,45.344,158.540
C06489=1029.216,168.068,391.442,169.108,45.346,158.540
C06490=1029.210,167.819,391.465,169.104,45.349,158.540
C06491=1029.205,167.569,391.487,169.101,45.351,158.540
C06492=1029.199,167.320,391.510,169.097,45.354,158.540
C06493=1029.192,167.072,391.533,169.095,45.356,158.540
C06494=1029.187,166.823,391.556,169.091,45.359,158.541
C06495=1029.181,166.574,391.579,169.088,45.361,158.541
C06496=1029.175,166.324,391.601,169.086,45.363,158.541
C06497=1029.169,166.076,391.623,169.082,45.366,158.541
C06498=1029.163,165.827,391.646,169.079,45.368,158.541
C06499=1029.158,165.579,391.669,169.076,45.371,158.541
C06500=1029.152,165.329,391.690,169.073,45.373,158.541
C06501=1029.146,165.081,391.713,169.070,45.375,158.542
C06502=1029.141,164.832,391.736,169.067,45.378,158.542
C06503=1029.135,164.583,391.759,169.064,45.381,158.542
C06504=1029.129,164.334,391.781,169.061,45.383,158.542
C06505=1029.123,164.085,391.804,169.058,45.385,158.542
C06506=1029.117,163.836,391.827,169.054,45.388,158.543
C06507=1029.112,163.586,391.849,169.052,45.390,158.543
C06508=1029.106,163.338,391.871,169.048,45.392,158.543
C06509=1029.100,163.090,391.894,169.046,45.394,158.543
C06510=1029.095,162.840,391.916,169.043,45.397,158.543
C06511=1029.088,162.591,391.938,169.039,45.400,158.543
C06512=1029.083,162.342,391.961,169.037,45.402,158.544
C06513=1029.077,162.093,391.984,169.033,45.404,158.544
C06514=1029.072,161.845,392.006,169.031,45.407,158.544
C06515=1029.066,161.596,392.028,169.027,45.409,158.544
C06516=1029.060,161.347,392.051,169.024,45.412,158.544
C06517=1029.055,161.097,392.073,169.022,45.414,158.544
C06518=1029.048,160.849,392.095,169.018,45.416,158.544
C06519=1029.043,160.600,392.118,169.016,45.419,158.545
C06520=1029.038,160.351,392.140,169.012,45.421,158.545
C06521=1029.032,160.102,392.163,169.009,45.424,158.545
C06522=1029.026,159.853,392.185,169.006,45.426,158.545
C06523=1029.020,159.604,392.208,169.003,45.429,158.545
C06524=1029.014,159.355,392.229,169.001,45.431,158.546
C06525=1029.009,159.106,392.252,168.997,45.434,158.546
C06526=1029.003,158.857,392.273,168.994,45.437,158.546
C06527=1028.996,158.608,392.295,168.991,45.439,158.546
C06528=1028.991,158.359,392.318,168.988,45.442,158.546
C06529=1028.984,158.110,392.340,168.985,45.445,158.547
C06530=1028.979,157.861,392.361,168.982,45.447,158.547
C06531=1028.972,157.613,392.383,168.979,45.449,158.547
C06532=1028.967,157.363,392.406,168.977,45.452,158.547
C06533=1028.961,157.114,392.427,168.973,45.454,158.547
C06534=1028.955,156.865,392.449,168.970,45.457,158.548
C06535=1028.948,156.581,392.474,168.967,45.460,158.548
C06536=1028.941,156.297,392.499,168.963,45.463,158.548
C06537=1028.935,156.013,392.524,168.960,45.466,158.548
C06538=1028.928,155.728,392.549,168.957,45.469,158.549
C06539=1028.922,155.480,392.571,168.954,45.472,158.549
C06540=1028.916,155.231,392.592,168.951,45.474,158.549
C06541=1028.910,154.982,392.615,168.948,45.477,158.549
C06542=1028.904,154.732,392.637,168.944,45.479,158.549
C06543=1028.899,154.484,392.658,168.942,45.482,158.550
C06544=1028.893,154.235,392.680,168.939,45.484,158.550
C06545=1028.887,153.985,392.702,168.936,45.487,158.550
C06546=1028.881,153.737,392.724,168.933,45.490,158.550
C06547=1028.875,153.488,392.746,168.931,45.492,158.550
C06548=1028.869,153.239,392.767,168.927,45.495,158.551
C06549=1028.863,152.990,392.789,168.924,45.498,158.551
C06550=1028.857,152.741,392.811,168.922,45.500,158.551
C06551=1028.851,152.492,392.832,168.918,45.503,158.551
C06552=1028.846,152.242,392.854,168.916,45.505,158.551
C06553=1028.839,151.993,392.876,168.913,45.508,158.552
C06554=1028.834,151.745,392.897,168.909,45.511,158.552
C06555=1028.828,151.496,392.919,168.907,45.513,158.552
C06556=1028.821,151.247,392.941,168.904,45.516,158.552
C06557=1028.815,150.998,392.963,168.901,45.519,158.553
C06558=1028.810,150.749,392.984,168.898,45.522,158.553
C06559=1028.803,150.500,393.006,168.895,45.524,158.553
C06560=1028.797,150.251,393.027,168.892,45.526,158.553
C06561=1028.792,150.002,393.049,168.889,45.529,158.553
C06562=1028.786,149.753,393.071,168.887,45.532,158.554
C06563=1028.780,149.504,393.092,168.883,45.534,158.554
C06564=1028.775,149.255,393.114,168.881,45.537,158.554
C06565=1028.768,149.006,393.135,168.878,45.540,158.554
C06566=1028.762,148.757,393.157,168.875,45.542,158.555
C06567=1028.757,148.508,393.178,168.872,45.545,158.555
C06568=1028.750,148.259,393.200,168.869,45.547,158.555
C06569=1028.745,148.010,393.220,168.866,45.550,158.555
C06570=1028.739,147.761,393.242,168.863,45.553,158.555
C06571=1028.733,147.511,393.264,168.861,45.556,158.556
C06572=1028.727,147.263,393.285,168.857,45.558,158.556
C06573=1028.721,147.014,393.306,168.855,45.561,158.556
C06574=1028.715,146.765,393.328,168.852,45.564,158.556
C06575=1028.709,146.516,393.349,168.849,45.566,158.556
C06576=1028.703,146.267,393.371,168.846,45.569,158.557
C06577=1028.698,146.018,393.392,168.843,45.571,158.557
C06578=1028.692,145.769,393.413,168.840,45.574,158.557
C06579=1028.686,145.519,393.435,168.838,45.577,158.557
C06580=1028.680,145.271,393.456,168.835,45.580,158.558
C06581=1028.673,145.022,393.477,168.831,45.583,158.558
C06582=1028.667,144.772,393.498,168.829,45.585,158.558
C06583=1028.662,144.524,393.519,168.826,45.588,158.558
C06584=1028.656,144.274,393.541,168.823,45.590,158.558
C06585=1028.650,144.026,393.562,168.820,45.593,158.559
C06586=1028.644,143.776,393.583,168.818,45.596,158.559
C06587=1028.638,143.528,393.604,168.814,45.599,158.559
C06588=1028.632,143.279,393.625,168.812,45.601,158.559
C06589=1028.626,143.029,393.646,168.809,45.604,158.560
C06590=1028.620,142.780,393.668,168.807,45.607,158.560
C06591=1028.614,142.531,393.689,168.803,45.609,158.560
C06592=1028.609,142.283,393.711,168.801,45.612,158.560
C06593=1028.602,142.033,393.731,168.798,45.615,158.561
C06594=1028.596,141.785,393.752,168.795,45.617,158.561
C06595=1028.590,141.535,393.774,168.792,45.620,158.561
C06596=1028.585,141.286,393.794,168.790,45.623,158.561
C06597=1028.579,141.037,393.816,168.786,45.626,158.562
C06598=1028.574,140.788,393.837,168.784,45.628,158.562
C06599=1028.566,140.503,393.861,168.781,45.632,158.562
C06600=1028.560,140.219,393.885,168.778,45.634,158.562
C06601=1028.552,139.934,393.909,168.774,45.637,158.563
C06602=1028.546,139.650,393.933,168.771,45.640,158.563
C06603=1028.540,139.401,393.954,168.768,45.643,158.563
C06604=1028.534,139.152,393.975,168.766,45.646,158.563
C06605=1028.529,138.903,393.996,168.762,45.649,158.563
C06606=1028.523,138.654,394.018,168.760,45.651,158.564
C06607=1028.517,138.405,394.038,168.757,45.654,158.564
C06608=1028.511,138.156,394.059,168.754,45.657,158.564
C06609=1028.505,137.907,394.079,168.751,45.660,158.565
C06610=1028.498,137.658,394.101,168.749,45.663,158.565
C06611=1028.493,137.408,394.121,168.745,45.665,158.565
C06612=1028.486,137.160,394.142,168.743,45.668,158.565
C06613=1028.481,136.910,394.163,168.740,45.671,158.565
C06614=1028.475,136.661,394.185,168.738,45.673,158.566
C06615=1028.469,136.412,394.205,168.734,45.676,158.566
C06616=1028.463,136.163,394.226,168.732,45.679,158.566
C06617=1028.457,135.914,394.247,168.729,45.682,158.566
C06618=1028.451,135.665,394.267,168.727,45.684,158.567
C06619=1028.445,135.416,394.288,168.723,45.687,158.567
C06620=1028.439,135.167,394.309,168.721,45.690,158.567
C06621=1028.433,134.917,394.329,168.718,45.693,158.567
C06622=1028.427,134.669,394.350,168.715,45.696,158.568
C06623=1028.421,134.419,394.371,168.712,45.699,158.568
C06624=1028.416,134.171,394.392,168.710,45.701,158.568
C06625=1028.409,133.921,394.412,168.707,45.704,158.568
C06626=1028.404,133.672,394.433,168.704,45.707,158.569
C06627=1028.397,133.423,394.454,168.701,45.710,158.569
C06628=1028.392,133.174,394.475,168.699,45.712,158.569
C06629=1028.386,132.925,394.495,168.696,45.714,158.569
C06630=1028.380,132.676,394.516,168.693,45.717,158.570
C06631=1028.374,132.427,394.536,168.691,45.720,158.570
C06632=1028.368,132.178,394.557,168.688,45.723,158.570
C06633=1028.362,131.928,394.578,168.685,45.726,158.570
C06634=1028.356,131.680,394.598,168.682,45.729,158.571
C06635=1028.350,131.430,394.619,168.680,45.731,158.571
C06636=1028.344,131.182,394.639,168.676,45.734,158.571
C06637=1028.339,130.933,394.660,168.674,45.737,158.571
C06638=1028.332,130.684,394.681,168.672,45.740,158.572
C06639=1028.327,130.435,394.701,168.669,45.743,158.572
C06640=1028.320,130.185,394.722,168.666,45.745,158.572
C06641=1028.314,129.936,394.742,168.663,45.748,158.572
C06642=1028.309,129.687,394.762,168.661,45.751,158.573
C06643=1028.302,129.438,394.783,168.658,45.754,158.573
C06644=1028.296,129.189,394.802,168.655,45.756,158.573
C06645=1028.290,128.940,394.824,168.652,45.759,158.573
C06646=1028.284,128.691,394.843,168.650,45.762,158.574
C06647=1028.278,128.442,394.864,168.647,45.766,158.574
C06648=1028.272,128.192,394.884,168.645,45.768,158.574
C06649=1028.266,127.944,394.904,168.641,45.771,158.574
C06650=1028.260,127.695,394.924,168.639,45.774,158.575
C06651=1028.254,127.445,394.945,168.636,45.777,158.575
C06652=1028.248,127.196,394.965,168.634,45.780,158.575
C06653=1028.242,126.947,394.985,168.630,45.783,158.575
C06654=1028.235,126.698,395.005,168.628,45.785,158.576
C06655=1028.229,126.449,395.025,168.625,45.788,158.576
C06656=1028.224,126.200,395.046,168.622,45.791,158.576
C06657=1028.217,125.950,395.066,168.619,45.794,158.576
C06658=1028.211,125.702,395.086,168.617,45.797,158.577
C06659=1028.205,125.453,395.106,168.615,45.800,158.577
C06660=1028.200,125.203,395.127,168.612,45.803,158.577
C06661=1028.194,124.954,395.147,168.609,45.805,158.578
C06662=1028.188,124.705,395.167,168.606,45.808,158.578
C06663=1028.180,124.421,395.190,168.603,45.811,158.578
C06664=1028.173,124.136,395.213,168.600,45.815,158.579
C06665=1028.166,123.851,395.236,168.597,45.818,158.579
C06666=1028.160,123.566,395.259,168.595,45.821,158.579
C06667=1028.154,123.318,395.279,168.591,45.824,158.579
C06668=1028.148,123.069,395.299,168.589,45.827,158.580
C06669=1028.142,122.818,395.319,168.586,45.830,158.580
C06670=1028.136,122.570,395.339,168.584,45.833,158.580
C06671=1028.130,122.321,395.359,168.580,45.835,158.580
C06672=1028.124,122.072,395.379,168.578,45.838,158.581
C06673=1028.118,121.822,395.400,168.576,45.841,158.581
C06674=1028.113,121.573,395.420,168.573,45.844,158.581
C06675=1028.107,121.325,395.440,168.570,45.847,158.581
C06676=1028.101,121.076,395.460,168.567,45.849,158.582
C06677=1028.094,120.826,395.480,168.565,45.852,158.582
C06678=1028.088,120.577,395.500,168.562,45.855,158.582
C06679=1028.083,120.328,395.520,168.559,45.858,158.582
C06680=1028.077,120.079,395.540,168.557,45.860,158.583
C06681=1028.071,119.830,395.560,168.554,45.863,158.583
C06682=1028.064,119.580,395.581,168.551,45.866,158.583
C06683=1028.059,119.331,395.600,168.549,45.869,158.583
C06684=1028.053,119.082,395.620,168.546,45.872,158.584
C06685=1028.047,118.833,395.640,168.544,45.874,158.584
C06686=1028.041,118.584,395.660,168.540,45.877,158.584
C06687=1028.035,118.335,395.681,168.538,45.881,158.585
C06688=1028.029,118.085,395.700,168.536,45.884,158.585
C06689=1028.023,117.837,395.720,168.533,45.886,158.585
C06690=1028.018,117.587,395.740,168.531,45.889,158.585
C06691=1028.012,117.339,395.760,168.528,45.892,158.586
C06692=1028.006,117.089,395.780,168.525,45.895,158.586
C06693=1028.000,116.840,395.800,168.523,45.898,158.586
C06694=1027.994,116.591,395.820,168.521,45.900,158.586
C06695=1027.988,116.341,395.839,168.517,45.903,158.587
C06696=1027.983,116.092,395.860,168.515,45.906,158.587
C06697=1027.977,115.843,395.880,168.512,45.909,158.587
C06698=1027.971,115.595,395.900,168.510,45.912,158.587
C06699=1027.965,115.345,395.919,168.507,45.914,158.588
C06700=1027.959,115.096,395.939,168.504,45.917,158.588
C06701=1027.952,114.847,395.959,168.502,45.919,158.588
C06702=1027.948,114.597,395.979,168.499,45.922,158.588
C06703=1027.942,114.348,395.999,168.496,45.925,158.589
C06704=1027.936,114.100,396.019,168.494,45.928,158.589
C06705=1027.930,113.850,396.038,168.492,45.930,158.589
C06706=1027.924,113.601,396.058,168.488,45.933,158.589
C06707=1027.918,113.352,396.078,168.486,45.936,158.590
C06708=1027.913,113.103,396.098,168.484,45.939,158.590
C06709=1027.907,112.854,396.118,168.482,45.941,158.590
C06710=1027.901,112.604,396.137,168.478,45.944,158.590
C06711=1027.895,112.355,396.157,168.476,45.947,158.591
C06712=1027.888,112.106,396.176,168.473,45.951,158.591
C06713=1027.882,111.857,396.196,168.471,45.953,158.591
C06714=1027.877,111.608,396.215,168.469,45.956,158.592
C06715=1027.871,111.359,396.235,168.465,45.959,158.592
C06716=1027.865,111.109,396.254,168.463,45.962,158.592
C06717=1027.859,110.861,396.274,168.461,45.964,158.592
C06718=1027.853,110.611,396.294,168.458,45.967,158.593
C06719=1027.847,110.362,396.314,168.455,45.970,158.593
C06720=1027.841,110.113,396.333,168.452,45.973,158.593
C06721=1027.834,109.863,396.352,168.450,45.976,158.593
C06722=1027.828,109.614,396.372,168.448,45.979,158.594
C06723=1027.823,109.365,396.391,168.445,45.982,158.594
C06724=1027.817,109.116,396.411,168.442,45.985,158.594
C06725=1027.810,108.867,396.430,168.439,45.988,158.594
C06726=1027.805,108.617,396.449,168.437,45.991,158.595
C06727=1027.798,108.333,396.472,168.434,45.994,158.595
C06728=1027.791,108.048,396.494,168.431,45.998,158.595
C06729=1027.784,107.763,396.515,168.428,46.001,158.596
C06730=1027.777,107.478,396.537,168.426,46.004,158.596
C06731=1027.771,107.229,396.557,168.422,46.007,158.596
C06732=1027.765,106.980,396.576,168.420,46.010,158.597
C06733=1027.759,106.731,396.595,168.418,46.013,158.597
C06734=1027.753,106.481,396.615,168.415,46.016,158.597
C06735=1027.746,106.233,396.634,168.413,46.019,158.597
C06736=1027.741,105.983,396.653,168.409,46.022,158.598
C06737=1027.735,105.734,396.672,168.407,46.025,158.598
C06738=1027.728,105.485,396.692,168.405,46.027,158.598
C06739=1027.723,105.236,396.711,168.402,46.030,158.598
C06740=1027.717,104.987,396.730,168.399,46.033,158.599
C06741=1027.711,104.737,396.750,168.397,46.036,158.599
C06742=1027.705,104.489,396.769,168.394,46.039,158.599
C06743=1027.699,104.239,396.788,168.392,46.042,158.600
C06744=1027.693,103.990,396.807,168.390,46.045,158.600
C06745=1027.687,103.741,396.826,168.386,46.048,158.600
C06746=1027.681,103.491,396.845,168.384,46.050,158.600
C06747=1027.675,103.242,396.865,168.382,46.053,158.601
C06748=1027.669,102.993,396.884,168.379,46.056,158.601
C06749=1027.663,102.744,396.903,168.377,46.060,158.601
C06750=1027.657,102.494,396.922,168.374,46.062,158.602
C06751=1027.651,102.245,396.941,168.371,46.065,158.602
C06752=1027.645,101.996,396.961,168.369,46.068,158.602
C06753=1027.639,101.747,396.980,168.367,46.071,158.602
C06754=1027.634,101.498,396.999,168.363,46.074,158.603
C06755=1027.628,101.249,397.018,168.361,46.076,158.603
C06756=1027.622,101.000,397.037,168.359,46.079,158.603
C06757=1027.616,100.750,397.056,168.356,46.082,158.603
C06758=1027.610,100.501,397.075,168.353,46.085,158.604
C06759=1027.604,100.252,397.094,168.351,46.088,158.604
C06760=1027.598,100.003,397.114,168.348,46.091,158.604
C06761=1027.592,99.754,397.133,168.346,46.094,158.605
C06762=1027.586,99.504,397.152,168.344,46.097,158.605
C06763=1027.580,99.255,397.171,168.340,46.100,158.605
C06764=1027.574,99.006,397.190,168.338,46.102,158.605
C06765=1027.568,98.757,397.208,168.336,46.106,158.606
C06766=1027.561,98.508,397.227,168.333,46.109,158.606
C06767=1027.555,98.258,397.246,168.331,46.111,158.606
C06768=1027.549,98.009,397.265,168.328,46.114,158.606
C06769=1027.544,97.760,397.283,168.325,46.118,158.607
C06770=1027.538,97.511,397.302,168.323,46.120,158.607
C06771=1027.531,97.261,397.320,168.320,46.123,158.607
C06772=1027.526,97.012,397.340,168.318,46.126,158.608
C06773=1027.519,96.763,397.358,168.315,46.129,158.608
C06774=1027.514,96.513,397.378,168.313,46.133,158.608
C06775=1027.507,96.264,397.396,168.310,46.135,158.608
C06776=1027.501,96.015,397.416,168.308,46.138,158.609
C06777=1027.495,95.766,397.434,168.305,46.141,158.609
C06778=1027.489,95.517,397.453,168.303,46.144,158.609
C06779=1027.483,95.268,397.472,168.301,46.147,158.610
C06780=1027.477,95.019,397.490,168.297,46.150,158.610
C06781=1027.471,94.769,397.508,168.295,46.153,158.610
C06782=1027.465,94.520,397.528,168.293,46.156,158.610
C06783=1027.459,94.271,397.546,168.290,46.159,158.611
C06784=1027.453,94.021,397.565,168.287,46.161,158.611
C06785=1027.447,93.772,397.584,168.285,46.165,158.611
C06786=1027.441,93.524,397.602,168.282,46.168,158.612
C06787=1027.435,93.274,397.622,168.280,46.170,158.612
C06788=1027.429,93.024,397.640,168.278,46.173,158.612
C06789=1027.423,92.775,397.659,168.274,46.176,158.612
C06790=1027.417,92.526,397.677,168.272,46.179,158.613
C06791=1027.411,92.242,397.699,168.269,46.183,158.613
C06792=1027.403,91.956,397.720,168.267,46.186,158.613
C06793=1027.397,91.672,397.741,168.264,46.189,158.614
C06794=1027.390,91.387,397.763,168.261,46.193,158.614
C06795=1027.384,91.138,397.782,168.259,46.195,158.614
C06796=1027.378,90.888,397.800,168.255,46.198,158.614
C06797=1027.372,90.640,397.818,168.253,46.201,158.615
C06798=1027.366,90.390,397.837,168.251,46.204,158.615
C06799=1027.360,90.141,397.856,168.249,46.206,158.615
C06800=1027.355,89.891,397.875,168.246,46.210,158.616
C06801=1027.348,89.642,397.893,168.244,46.213,158.616
C06802=1027.342,89.394,397.911,168.241,46.216,158.616
C06803=1027.336,89.144,397.929,168.238,46.219,158.616
C06804=1027.330,88.895,397.948,168.236,46.222,158.617
C06805=1027.323,88.646,397.967,168.234,46.225,158.617
C06806=1027.318,88.395,397.985,168.231,46.228,158.617
C06807=1027.312,88.147,398.004,168.228,46.230,158.617
C06808=1027.306,87.897,398.021,168.225,46.234,158.618
C06809=1027.300,87.648,398.040,168.223,46.237,158.618
C06810=1027.293,87.398,398.058,168.221,46.240,158.618
C06811=1027.287,87.149,398.077,168.218,46.243,158.619
C06812=1027.281,86.901,398.095,168.216,46.246,158.619
C06813=1027.275,86.651,398.113,168.214,46.249,158.619
C06814=1027.269,86.402,398.132,168.210,46.252,158.619
C06815=1027.262,86.152,398.149,168.208,46.254,158.620
C06816=1027.257,85.904,398.168,168.206,46.258,158.620
C06817=1027.251,85.654,398.186,168.203,46.261,158.620
C06818=1027.245,85.405,398.205,168.201,46.264,158.621
C06819=1027.239,85.155,398.223,168.198,46.266,158.621
C06820=1027.233,84.907,398.241,168.195,46.270,158.621
C06821=1027.227,84.657,398.259,168.193,46.273,158.622
C06822=1027.220,84.408,398.278,168.191,46.276,158.622
C06823=1027.215,84.159,398.295,168.188,46.279,158.622
C06824=1027.208,83.910,398.314,168.186,46.282,158.622
C06825=1027.202,83.660,398.332,168.183,46.285,158.623
C06826=1027.196,83.411,398.351,168.180,46.288,158.623
C06827=1027.190,83.162,398.368,168.178,46.290,158.623
C06828=1027.184,82.913,398.387,168.176,46.293,158.623
C06829=1027.178,82.663,398.405,168.174,46.297,158.624
C06830=1027.172,82.414,398.423,168.171,46.300,158.624
C06831=1027.166,82.165,398.441,168.168,46.302,158.624
C06832=1027.160,81.915,398.460,168.166,46.305,158.625
C06833=1027.155,81.666,398.478,168.163,46.308,158.625
C06834=1027.149,81.416,398.496,168.161,46.312,158.625
C06835=1027.142,81.167,398.514,168.159,46.314,158.626
C06836=1027.137,80.918,398.532,168.155,46.317,158.626
C06837=1027.130,80.669,398.551,168.153,46.320,158.626
C06838=1027.124,80.419,398.568,168.151,46.323,158.626
C06839=1027.119,80.170,398.586,168.148,46.326,158.626
C06840=1027.112,79.921,398.605,168.146,46.329,158.627
C06841=1027.106,79.671,398.623,168.144,46.332,158.627
C06842=1027.100,79.423,398.641,168.141,46.335,158.627
C06843=1027.094,79.173,398.659,168.138,46.338,158.628
C06844=1027.088,78.924,398.677,168.136,46.340,158.628
C06845=1027.082,78.675,398.695,168.134,46.343,158.628
C06846=1027.076,78.425,398.713,168.130,46.346,158.628
C06847=1027.070,78.176,398.731,168.128,46.350,158.629
C06848=1027.064,77.927,398.749,168.126,46.352,158.629
C06849=1027.058,77.677,398.767,168.124,46.355,158.629
C06850=1027.052,77.428,398.785,168.121,46.358,158.630
C06851=1027.046,77.179,398.803,168.118,46.361,158.630
C06852=1027.040,76.930,398.821,168.116,46.364,158.630
C06853=1027.034,76.681,398.839,168.113,46.367,158.630
C06854=1027.028,76.431,398.857,168.111,46.370,158.631
C06855=1027.022,76.146,398.877,168.108,46.374,158.631
C06856=1027.014,75.861,398.898,168.105,46.377,158.631
C06857=1027.008,75.576,398.918,168.103,46.380,158.632
C06858=1027.001,75.292,398.938,168.100,46.384,158.632
C06859=1026.994,75.042,398.956,168.097,46.387,158.632
C06860=1026.989,74.793,398.973,168.095,46.390,158.633
C06861=1026.982,74.544,398.991,168.092,46.393,158.633
C06862=1026.976,74.294,399.009,168.090,46.396,158.633
C06863=1026.970,74.046,399.027,168.087,46.399,158.633
C06864=1026.964,73.796,399.045,168.085,46.402,158.634
C06865=1026.958,73.547,399.062,168.083,46.405,158.634
C06866=1026.952,73.297,399.080,168.080,46.408,158.634
C06867=1026.946,73.047,399.098,168.077,46.411,158.635
C06868=1026.940,72.799,399.115,168.075,46.413,158.635
C06869=1026.933,72.549,399.133,168.072,46.417,158.635
C06870=1026.928,72.300,399.151,168.070,46.420,158.635
C06871=1026.922,72.050,399.169,168.068,46.423,158.636
C06872=1026.915,71.802,399.186,168.064,46.426,158.636
C06873=1026.909,71.552,399.204,168.062,46.429,158.636
C06874=1026.904,71.303,399.222,168.060,46.432,158.637
C06875=1026.898,71.054,399.240,168.057,46.435,158.637
C06876=1026.891,70.805,399.257,168.055,46.438,158.637
C06877=1026.885,70.555,399.275,168.053,46.440,158.637
C06878=1026.880,70.306,399.292,168.050,46.444,158.638
C06879=1026.874,70.056,399.310,168.047,46.447,158.638
C06880=1026.867,69.808,399.327,168.045,46.450,158.638
C06881=1026.861,69.558,399.345,168.043,46.452,158.638
C06882=1026.856,69.309,399.363,168.040,46.455,158.639
C06883=1026.849,69.059,399.380,168.038,46.459,158.639
C06884=1026.843,68.810,399.397,168.036,46.462,158.639
C06885=1026.837,68.561,399.415,168.032,46.465,158.640
C06886=1026.831,68.312,399.432,168.030,46.467,158.640
C06887=1026.825,68.062,399.450,168.028,46.471,158.640
C06888=1026.820,67.812,399.467,168.025,46.474,158.640
C06889=1026.813,67.563,399.484,168.023,46.477,158.641
C06890=1026.807,67.314,399.502,168.020,46.479,158.641
C06891=1026.800,67.065,399.519,168.017,46.483,158.641
C06892=1026.795,66.815,399.537,168.015,46.486,158.642
C06893=1026.789,66.566,399.555,168.013,46.489,158.642
C06894=1026.782,66.317,399.572,168.010,46.492,158.642
C06895=1026.776,66.067,399.590,168.008,46.495,158.642
C06896=1026.770,65.818,399.606,168.006,46.498,158.643
C06897=1026.764,65.568,399.624,168.002,46.501,158.643
C06898=1026.758,65.319,399.641,168.000,46.504,158.643
C06899=1026.752,65.070,399.659,167.998,46.507,158.644
C06900=1026.746,64.821,399.676,167.995,46.510,158.644
C06901=1026.739,64.571,399.694,167.993,46.513,158.644
C06902=1026.733,64.322,399.710,167.991,46.516,158.644
C06903=1026.728,64.073,399.728,167.988,46.519,158.645
C06904=1026.721,63.823,399.745,167.985,46.522,158.645
C06905=1026.716,63.574,399.763,167.983,46.525,158.645
C06906=1026.709,63.325,399.780,167.981,46.528,158.645
C06907=1026.704,63.075,399.797,167.978,46.531,158.646
C06908=1026.697,62.826,399.814,167.976,46.534,158.646
C06909=1026.690,62.577,399.831,167.972,46.537,158.646
C06910=1026.685,62.327,399.848,167.971,46.541,158.647
C06911=1026.678,62.078,399.865,167.968,46.543,158.647
C06912=1026.672,61.829,399.881,167.965,46.547,158.647
C06913=1026.666,61.579,399.899,167.963,46.550,158.648
C06914=1026.660,61.330,399.916,167.960,46.553,158.648
C06915=1026.653,61.080,399.933,167.958,46.556,158.648
C06916=1026.647,60.831,399.950,167.956,46.559,158.648
C06917=1026.640,60.582,399.967,167.953,46.563,158.649
C06918=1026.634,60.333,399.984,167.951,46.565,158.649
C06919=1026.628,60.047,400.003,167.948,46.569,158.649
C06920=1026.621,59.763,400.023,167.945,46.573,158.650
C06921=1026.613,59.478,400.042,167.941,46.576,158.650
C06922=1026.607,59.192,400.062,167.938,46.580,158.650
C06923=1026.600,58.944,400.079,167.937,46.583,158.651
C06924=1026.594,58.694,400.095,167.934,46.586,158.651
C06925=1026.587,58.445,400.112,167.931,46.589,158.651
C06926=1026.582,58.195,400.129,167.929,46.592,158.652
C06927=1026.575,57.946,400.147,167.927,46.595,158.652
C06928=1026.569,57.696,400.163,167.924,46.598,158.652
C06929=1026.563,57.448,400.180,167.922,46.602,158.652
C06930=1026.557,57.198,400.196,167.920,46.604,158.653
C06931=1026.551,56.949,400.214,167.916,46.607,158.653
C06932=1026.545,56.699,400.231,167.914,46.611,158.653
C06933=1026.538,56.450,400.248,167.911,46.614,158.653
C06934=1026.532,56.200,400.264,167.909,46.617,158.654
C06935=1026.526,55.951,400.281,167.907,46.619,158.654
C06936=1026.520,55.701,400.298,167.904,46.623,158.654
C06937=1026.514,55.453,400.315,167.901,46.626,158.655
C06938=1026.507,55.203,400.332,167.899,46.629,158.655
C06939=1026.501,54.954,400.349,167.896,46.632,158.655
C06940=1026.496,54.704,400.365,167.894,46.635,158.655
C06941=1026.490,54.455,400.382,167.892,46.638,158.656
C06942=1026.483,54.205,400.399,167.889,46.641,158.656
C06943=1026.477,53.956,400.415,167.887,46.644,158.656
C06944=1026.471,53.707,400.432,167.885,46.647,158.657
C06945=1026.465,53.457,400.449,167.881,46.650,158.657
C06946=1026.459,53.208,400.466,167.879,46.653,158.657
C06947=1026.453,52.959,400.483,167.877,46.656,158.657
C06948=1026.446,52.709,400.499,167.874,46.660,158.658
C06949=1026.440,52.460,400.516,167.872,46.662,158.658
C06950=1026.435,52.210,400.533,167.869,46.665,158.658
C06951=1026.429,51.962,400.550,167.867,46.669,158.659
C06952=1026.422,51.712,400.567,167.864,46.672,158.659
C06953=1026.416,51.462,400.583,167.862,46.674,158.659
C06954=1026.410,51.214,400.600,167.859,46.677,158.659
C06955=1026.405,50.964,400.617,167.857,46.681,158.660
C06956=1026.398,50.714,400.633,167.855,46.684,158.660
C06957=1026.392,50.465,400.650,167.851,46.687,158.660
C06958=1026.386,50.216,400.667,167.849,46.689,158.660
C06959=1026.380,49.966,400.683,167.847,46.692,158.661
C06960=1026.374,49.717,400.700,167.844,46.696,158.661
C06961=1026.368,49.467,400.717,167.842,46.699,158.661
C06962=1026.362,49.218,400.733,167.840,46.702,158.662
C06963=1026.356,48.969,400.750,167.836,46.705,158.662
C06964=1026.350,48.720,400.767,167.834,46.707,158.662
C06965=1026.344,48.470,400.784,167.832,46.711,158.662
C06966=1026.338,48.220,400.800,167.829,46.714,158.663
C06967=1026.332,47.972,400.817,167.827,46.717,158.663
C06968=1026.326,47.722,400.833,167.825,46.719,158.663
C06969=1026.320,47.473,400.850,167.821,46.722,158.663
C06970=1026.314,47.224,400.867,167.819,46.725,158.664
C06971=1026.308,46.974,400.884,167.817,46.729,158.664
C06972=1026.302,46.724,400.900,167.815,46.732,158.664
C06973=1026.296,46.475,400.916,167.812,46.735,158.664
C06974=1026.290,46.226,400.933,167.810,46.737,158.665
C06975=1026.284,45.977,400.949,167.807,46.740,158.665
C06976=1026.278,45.727,400.966,167.804,46.743,158.665
C06977=1026.272,45.477,400.983,167.802,46.746,158.665
C06978=1026.266,45.228,400.999,167.800,46.749,158.666
C06979=1026.260,44.979,401.015,167.797,46.753,158.666
C06980=1026.254,44.730,401.032,167.795,46.755,158.666
C06981=1026.248,44.480,401.049,167.792,46.758,158.666
C06982=1026.243,44.231,401.066,167.789,46.761,158.667
C06983=1026.235,43.946,401.085,167.787,46.764,158.667
C06984=1026.229,43.660,401.103,167.784,46.768,158.667
C06985=1026.222,43.375,401.122,167.781,46.771,158.668
C06986=1026.216,43.090,401.141,167.778,46.774,158.668
C06987=1026.209,42.840,401.157,167.776,46.777,158.668
C06988=1026.203,42.591,401.174,167.773,46.780,158.668
C06989=1026.197,42.341,401.191,167.770,46.784,158.669
C06990=1026.191,42.092,401.207,167.768,46.787,158.669
C06991=1026.185,41.843,401.223,167.766,46.789,158.669
C06992=1026.179,41.593,401.239,167.763,46.792,158.669
C06993=1026.173,41.344,401.256,167.761,46.796,158.670
C06994=1026.166,41.095,401.271,167.759,46.799,158.670
C06995=1026.160,40.845,401.288,167.755,46.802,158.670
C06996=1026.154,40.596,401.304,167.753,46.804,158.670
C06997=1026.148,40.346,401.320,167.751,46.808,158.671
C06998=1026.142,40.096,401.336,167.748,46.811,158.671
C06999=1026.136,39.847,401.352,167.746,46.814,158.671
C07000=1026.130,39.598,401.368,167.743,46.817,158.671
C07001=1026.124,39.348,401.385,167.740,46.820,158.672
C07002=1026.118,39.099,401.401,167.739,46.823,158.672
C07003=1026.112,38.850,401.417,167.735,46.826,158.672
C07004=1026.106,38.601,401.433,167.733,46.829,158.673
C07005=1026.100,38.351,401.449,167.731,46.832,158.673
C07006=1026.094,38.102,401.465,167.728,46.835,158.673
C07007=1026.088,37.853,401.482,167.726,46.838,158.673
C07008=1026.082,37.603,401.498,167.724,46.841,158.674
C07009=1026.076,37.354,401.514,167.720,46.844,158.674
C07010=1026.069,37.104,401.531,167.718,46.847,158.674
C07011=1026.063,36.854,401.546,167.716,46.850,158.674
C07012=1026.057,36.605,401.562,167.713,46.854,158.675
C07013=1026.051,36.355,401.578,167.711,46.856,158.675
C07014=1026.044,36.106,401.594,167.708,46.859,158.675
C07015=1026.039,35.857,401.610,167.706,46.863,158.676
C07016=1026.033,35.607,401.626,167.703,46.866,158.676
C07017=1026.026,35.358,401.641,167.700,46.869,158.676
C07018=1026.020,35.109,401.658,167.698,46.872,158.676
C07019=1026.014,34.859,401.674,167.695,46.875,158.677
C07020=1026.008,34.610,401.689,167.693,46.878,158.677
C07021=1026.002,34.360,401.705,167.691,46.881,158.677
C07022=1025.996,34.111,401.721,167.688,46.885,158.677
C07023=1025.990,33.861,401.736,167.685,46.887,158.678
C07024=1025.984,33.612,401.752,167.682,46.890,158.678
C07025=1025.978,33.363,401.769,167.680,46.893,158.678
C07026=1025.971,33.114,401.784,167.678,46.897,158.679
C07027=1025.965,32.864,401.800,167.675,46.900,158.679
C07028=1025.959,32.615,401.816,167.673,46.903,158.679
C07029=1025.953,32.365,401.832,167.669,46.906,158.679
C07030=1025.947,32.115,401.847,167.668,46.909,158.680
C07031=1025.940,31.866,401.863,167.665,46.912,158.680
C07032=1025.934,31.617,401.879,167.662,46.915,158.680
C07033=1025.929,31.367,401.895,167.660,46.918,158.680
C07034=1025.922,31.118,401.911,167.657,46.922,158.681
C07035=1025.916,30.869,401.927,167.655,46.924,158.681
C07036=1025.911,30.619,401.942,167.653,46.927,158.681
C07037=1025.904,30.370,401.958,167.649,46.930,158.681
C07038=1025.898,30.120,401.974,167.647,46.934,158.682
C07039=1025.891,29.871,401.989,167.645,46.937,158.682
C07040=1025.886,29.622,402.005,167.642,46.940,158.682
C07041=1025.880,29.372,402.021,167.640,46.942,158.682
C07042=1025.874,29.123,402.036,167.637,46.945,158.683
C07043=1025.868,28.873,402.052,167.635,46.949,158.683
C07044=1025.862,28.624,402.068,167.632,46.952,158.683
C07045=1025.856,28.375,402.084,167.629,46.955,158.683
C07046=1025.850,28.125,402.099,167.627,46.958,158.684
C07047=1025.842,27.839,402.117,167.624,46.961,158.684
C07048=1025.836,27.554,402.135,167.621,46.964,158.684
C07049=1025.829,27.269,402.153,167.618,46.968,158.684
C07050=1025.822,26.984,402.171,167.615,46.972,158.685
C07051=1025.815,26.734,402.186,167.613,46.975,158.685
C07052=1025.809,26.485,402.202,167.610,46.979,158.685
C07053=1025.803,26.235,402.217,167.608,46.981,158.686
C07054=1025.797,25.985,402.233,167.605,46.984,158.686
C07055=1025.791,25.736,402.248,167.602,46.987,158.686
C07056=1025.786,25.487,402.263,167.600,46.991,158.686
C07057=1025.779,25.238,402.279,167.597,46.994,158.687
C07058=1025.773,24.988,402.294,167.595,46.997,158.687
C07059=1025.767,24.738,402.310,167.592,47.000,158.687
C07060=1025.760,24.489,402.325,167.590,47.003,158.687
C07061=1025.754,24.239,402.340,167.588,47.006,158.688
C07062=1025.748,23.990,402.356,167.584,47.009,158.688
C07063=1025.742,23.740,402.371,167.582,47.013,158.688
C07064=1025.737,23.491,402.386,167.579,47.016,158.688
C07065=1025.730,23.242,402.402,167.577,47.018,158.689
C07066=1025.723,22.992,402.417,167.574,47.022,158.689
C07067=1025.718,22.743,402.433,167.572,47.025,158.689
C07068=1025.711,22.493,402.448,167.570,47.028,158.690
C07069=1025.705,22.244,402.464,167.566,47.031,158.690
C07070=1025.700,21.995,402.478,167.564,47.034,158.690
C07071=1025.693,21.746,402.494,167.561,47.037,158.690
C07072=1025.687,21.496,402.510,167.559,47.040,158.691
C07073=1025.681,21.246,402.525,167.556,47.043,158.691
C07074=1025.675,20.996,402.540,167.554,47.046,158.691
C07075=1025.669,20.748,402.555,167.552,47.049,158.691
C07076=1025.663,20.498,402.570,167.549,47.053,158.692
C07077=1025.657,20.248,402.586,167.546,47.056,158.692
C07078=1025.651,19.999,402.602,167.543,47.059,158.692
C07079=1025.644,19.749,402.616,167.541,47.062,158.692
C07080=1025.639,19.500,402.632,167.538,47.065,158.692
C07081=1025.633,19.250,402.647,167.536,47.068,158.693
C07082=1025.626,19.001,402.662,167.534,47.071,158.693
C07083=1025.620,18.752,402.677,167.530,47.074,158.693
C07084=1025.614,18.502,402.693,167.528,47.077,158.694
C07085=1025.608,18.253,402.707,167.525,47.081,158.694
C07086=1025.602,18.003,402.722,167.523,47.083,158.694
C07087=1025.595,17.753,402.737,167.520,47.086,158.694
C07088=1025.590,17.503,402.753,167.518,47.089,158.695
C07089=1025.584,17.255,402.768,167.515,47.093,158.695
C07090=1025.577,17.005,402.783,167.513,47.096,158.695
C07091=1025.571,16.756,402.798,167.509,47.099,158.695
C07092=1025.565,16.506,402.813,167.507,47.102,158.696
C07093=1025.560,16.257,402.828,167.505,47.105,158.696
C07094=1025.553,16.007,402.843,167.502,47.108,158.696
C07095=1025.547,15.758,402.858,167.500,47.111,158.696
C07096=1025.540,15.508,402.873,167.497,47.114,158.696
C07097=1025.535,15.259,402.888,167.495,47.118,158.697
C07098=1025.529,15.009,402.903,167.492,47.121,158.697
C07099=1025.523,14.759,402.918,167.489,47.124,158.697
C07100=1025.516,14.511,402.933,167.486,47.127,158.697
C07101=1025.510,14.261,402.948,167.484,47.130,158.698
C07102=1025.504,14.011,402.964,167.482,47.133,158.698
C07103=1025.498,13.762,402.979,167.479,47.136,158.698
C07104=1025.492,13.513,402.993,167.477,47.139,158.699
C07105=1025.486,13.263,403.008,167.473,47.142,158.699
C07106=1025.480,13.013,403.022,167.472,47.146,158.699
C07107=1025.474,12.764,403.037,167.468,47.149,158.699
C07108=1025.468,12.514,403.052,167.466,47.152,158.700
C07109=1025.461,12.265,403.067,167.463,47.155,158.700
C07110=1025.456,12.016,403.082,167.460,47.158,158.700
C07111=1025.448,11.731,403.098,167.457,47.162,158.700
C07112=1025.441,11.448,403.115,167.454,47.166,158.701
C07113=1025.434,11.163,403.132,167.451,47.170,158.701
C07114=1025.427,10.880,403.148,167.448,47.173,158.701
C07115=1025.420,10.630,403.163,167.446,47.176,158.702
C07116=1025.414,10.381,403.178,167.443,47.179,158.702
C07117=1025.408,10.132,403.193,167.441,47.182,158.702
C07118=1025.402,9.881,403.207,167.438,47.186,158.702
C07119=1025.396,9.632,403.222,167.436,47.189,158.703
C07120=1025.390,9.383,403.236,167.432,47.192,158.703
C07121=1025.384,9.133,403.251,167.430,47.196,158.703
C07122=1025.378,8.884,403.266,167.427,47.199,158.703
C07123=1025.371,8.635,403.281,167.425,47.201,158.704
C07124=1025.365,8.385,403.295,167.422,47.205,158.704
C07125=1025.359,8.136,403.309,167.420,47.208,158.704
C07126=1025.352,7.886,403.324,167.417,47.211,158.704
C07127=1025.347,7.637,403.339,167.415,47.214,158.705
C07128=1025.341,7.387,403.353,167.412,47.218,158.705
C07129=1025.334,7.137,403.368,167.409,47.221,158.705
C07130=1025.328,6.888,403.382,167.406,47.224,158.705
C07131=1025.322,6.638,403.397,167.404,47.227,158.706
C07132=1025.317,6.389,403.411,167.401,47.230,158.706
C07133=1025.310,6.139,403.426,167.399,47.233,158.706
C07134=1025.304,5.890,403.441,167.396,47.236,158.706
C07135=1025.298,5.641,403.456,167.394,47.239,158.707
C07136=1025.292,5.390,403.470,167.391,47.243,158.707
C07137=1025.285,5.142,403.484,167.388,47.246,158.707
C07138=1025.279,4.892,403.499,167.385,47.249,158.707
C07139=1025.274,4.642,403.513,167.383,47.252,158.708
C07140=1025.267,4.393,403.528,167.380,47.255,158.708
C07141=1025.261,4.144,403.542,167.378,47.258,158.708
C07142=1025.255,3.894,403.557,167.375,47.261,158.708
C07143=1025.250,3.645,403.571,167.372,47.264,158.708
C07144=1025.243,3.395,403.586,167.369,47.267,158.709
C07145=1025.237,3.145,403.600,167.367,47.271,158.709
C07146=1025.231,2.896,403.615,167.364,47.274,158.709
C07147=1025.224,2.646,403.629,167.362,47.277,158.709
C07148=1025.219,2.397,403.643,167.359,47.280,158.710
C07149=1025.212,2.147,403.658,167.357,47.283,158.710
C07150=1025.207,1.898,403.672,167.353,47.286,158.710
C07151=1025.200,1.648,403.687,167.351,47.289,158.710
C07152=1025.195,1.399,403.701,167.348,47.292,158.711
C07153=1025.189,1.149,403.716,167.346,47.295,158.711
C07154=1025.183,0.900,403.730,167.343,47.298,158.711
C07155=1025.177,0.650,403.744,167.341,47.301,158.711
C07156=1025.171,0.400,403.759,167.337,47.304,158.711
C07157=1025.165,0.151,403.772,167.336,47.308,158.712
C07158=1025.158,-0.098,403.787,167.332,47.311,158.712
C07159=1025.153,-0.347,403.802,167.330,47.314,158.712
C07160=1025.146,-0.598,403.816,167.327,47.317,158.712
C07161=1025.141,-0.847,403.831,167.325,47.320,158.713
C07162=1025.135,-1.097,403.845,167.322,47.323,158.713
C07163=1025.129,-1.346,403.859,167.319,47.326,158.713
C07164=1025.123,-1.595,403.873,167.316,47.329,158.713
C07165=1025.117,-1.845,403.888,167.314,47.332,158.714
C07166=1025.111,-2.094,403.902,167.311,47.335,158.714
C07167=1025.104,-2.344,403.916,167.309,47.338,158.714
C07168=1025.099,-2.594,403.930,167.306,47.341,158.714
C07169=1025.093,-2.843,403.945,167.304,47.344,158.714
C07170=1025.087,-3.093,403.959,167.300,47.347,158.715
C07171=1025.081,-3.342,403.974,167.298,47.350,158.715
C07172=1025.075,-3.592,403.988,167.295,47.353,158.715
C07173=1025.070,-3.842,404.002,167.293,47.356,158.715
C07174=1025.063,-4.091,404.016,167.290,47.360,158.716
C07175=1025.056,-4.368,404.032,167.287,47.363,158.716
C07176=1025.050,-4.646,404.047,167.284,47.367,158.716
C07177=1025.043,-4.923,404.063,167.281,47.371,158.716
C07178=1025.036,-5.200,404.077,167.278,47.374,158.716
C07179=1025.029,-5.454,404.092,167.276,47.377,158.717
C07180=1025.024,-5.709,404.107,167.272,47.380,158.717
C07181=1025.017,-5.963,404.121,167.269,47.384,158.717
C07182=1025.011,-6.218,404.135,167.267,47.387,158.718
C07183=1025.005,-6.466,404.149,167.264,47.390,158.718
C07184=1024.999,-6.717,404.163,167.261,47.393,158.718
C07185=1024.992,-6.966,404.176,167.259,47.397,158.718
C07186=1024.987,-7.216,404.190,167.256,47.400,158.718
C07187=1024.980,-7.465,404.204,167.254,47.403,158.719
C07188=1024.974,-7.714,404.218,167.250,47.406,158.719
C07189=1024.967,-7.964,404.232,167.248,47.410,158.719
C07190=1024.962,-8.214,404.246,167.245,47.413,158.719
C07191=1024.956,-8.463,404.259,167.242,47.416,158.720
C07192=1024.949,-8.713,404.274,167.240,47.419,158.720
C07193=1024.943,-8.962,404.287,167.237,47.422,158.720
C07194=1024.938,-9.212,404.301,167.234,47.425,158.720
C07195=1024.932,-9.461,404.315,167.232,47.428,158.721
C07196=1024.925,-9.711,404.329,167.228,47.431,158.721
C07197=1024.920,-9.961,404.342,167.227,47.435,158.721
C07198=1024.913,-10.210,404.356,167.223,47.438,158.721
C07199=1024.907,-10.460,404.371,167.221,47.441,158.721
C07200=1024.901,-10.709,404.384,167.218,47.444,158.722
C07201=1024.896,-10.959,404.398,167.215,47.448,158.722
C07202=1024.889,-11.209,404.411,167.213,47.451,158.722
C07203=1024.883,-11.458,404.425,167.210,47.454,158.722
C07204=1024.877,-11.707,404.439,167.208,47.457,158.723
C07205=1024.872,-11.957,404.452,167.204,47.460,158.723
C07206=1024.865,-12.207,404.466,167.201,47.464,158.723
C07207=1024.859,-12.457,404.480,167.199,47.466,158.723
C07208=1024.853,-12.705,404.494,167.196,47.470,158.723
C07209=1024.847,-12.955,404.508,167.194,47.472,158.724
C07210=1024.841,-13.205,404.521,167.191,47.476,158.724
C07211=1024.835,-13.454,404.535,167.189,47.479,158.724
C07212=1024.829,-13.704,404.549,167.186,47.482,158.724
C07213=1024.823,-13.953,404.562,167.182,47.485,158.725
C07214=1024.817,-14.202,404.576,167.180,47.488,158.725
C07215=1024.811,-14.453,404.590,167.177,47.491,158.725
C07216=1024.805,-14.702,404.603,167.175,47.494,158.725
C07217=1024.799,-14.952,404.617,167.172,47.497,158.725
C07218=1024.793,-15.201,404.630,167.169,47.501,158.726
C07219=1024.787,-15.451,404.645,167.167,47.504,158.726
C07220=1024.781,-15.700,404.658,167.163,47.507,158.726
C07221=1024.775,-15.950,404.671,167.161,47.510,158.726
C07222=1024.770,-16.200,404.684,167.158,47.514,158.727
C07223=1024.763,-16.449,404.697,167.155,47.517,158.727
C07224=1024.757,-16.699,404.711,167.153,47.520,158.727
C07225=1024.750,-16.948,404.724,167.150,47.523,158.727
C07226=1024.744,-17.198,404.738,167.147,47.527,158.727
C07227=1024.739,-17.447,404.752,167.145,47.530,158.728
C07228=1024.733,-17.697,404.764,167.141,47.533,158.728
C07229=1024.726,-17.947,404.778,167.138,47.537,158.728
C07230=1024.720,-18.196,404.791,167.136,47.539,158.728
C07231=1024.714,-18.446,404.805,167.133,47.543,158.729
C07232=1024.708,-18.695,404.818,167.130,47.546,158.729
C07233=1024.702,-18.945,404.831,167.128,47.549,158.729
C07234=1024.696,-19.194,404.844,167.125,47.552,158.729
C07235=1024.690,-19.444,404.858,167.122,47.555,158.729
C07236=1024.684,-19.694,404.871,167.120,47.559,158.730
C07237=1024.677,-19.943,404.885,167.117,47.562,158.730
C07238=1024.671,-20.193,404.897,167.114,47.565,158.730
C07239=1024.665,-20.473,404.913,167.110,47.569,158.730
C07240=1024.658,-20.753,404.927,167.107,47.572,158.731
C07241=1024.651,-21.034,404.942,167.104,47.576,158.731
C07242=1024.645,-21.315,404.957,167.101,47.580,158.731
C07243=1024.639,-21.564,404.970,167.098,47.583,158.731
C07244=1024.633,-21.813,404.983,167.096,47.586,158.732
C07245=1024.626,-22.063,404.997,167.093,47.589,158.732
C07246=1024.620,-22.313,405.010,167.091,47.592,158.732
C07247=1024.614,-22.562,405.023,167.088,47.596,158.732
C07248=1024.608,-22.812,405.037,167.085,47.599,158.732
C07249=1024.602,-23.062,405.049,167.082,47.602,158.733
C07250=1024.596,-23.311,405.063,167.079,47.605,158.733
C07251=1024.591,-23.560,405.076,167.076,47.609,158.733
C07252=1024.585,-23.810,405.089,167.074,47.612,158.733
C07253=1024.578,-24.060,405.102,167.071,47.615,158.733
C07254=1024.572,-24.309,405.115,167.068,47.618,158.734
C07255=1024.566,-24.559,405.128,167.066,47.621,158.734
C07256=1024.560,-24.808,405.141,167.062,47.624,158.734
C07257=1024.555,-25.058,405.154,167.059,47.628,158.734
C07258=1024.549,-25.307,405.168,167.057,47.631,158.735
C07259=1024.543,-25.557,405.180,167.054,47.634,158.735
C07260=1024.537,-25.807,405.194,167.051,47.637,158.735
C07261=1024.530,-26.056,405.207,167.049,47.640,158.735
C07262=1024.525,-26.306,405.220,167.046,47.643,158.735
C07263=1024.519,-26.555,405.233,167.044,47.646,158.736
C07264=1024.513,-26.805,405.246,167.040,47.650,158.736
C07265=1024.507,-27.054,405.259,167.037,47.653,158.736
C07266=1024.501,-27.304,405.272,167.035,47.656,158.736
C07267=1024.495,-27.554,405.285,167.032,47.659,158.736
C07268=1024.489,-27.804,405.297,167.029,47.663,158.737
C07269=1024.483,-28.053,405.311,167.026,47.666,158.737
C07270=1024.477,-28.303,405.323,167.024,47.669,158.737
C07271=1024.471,-28.553,405.336,167.021,47.672,158.737
C07272=1024.465,-28.802,405.349,167.018,47.676,158.737
C07273=1024.459,-29.052,405.362,167.015,47.678,158.738
C07274=1024.452,-29.301,405.375,167.012,47.682,158.738
C07275=1024.447,-29.551,405.387,167.009,47.685,158.738
C07276=1024.441,-29.801,405.400,167.006,47.689,158.738
C07277=1024.434,-30.050,405.413,167.004,47.691,158.738
C07278=1024.429,-30.300,405.426,167.001,47.695,158.739
C07279=1024.423,-30.550,405.438,166.998,47.698,158.739
C07280=1024.416,-30.799,405.451,166.995,47.702,158.739
C07281=1024.410,-31.049,405.464,166.992,47.704,158.739
C07282=1024.404,-31.298,405.476,166.990,47.708,158.740
C07283=1024.398,-31.547,405.489,166.986,47.711,158.740
